LIN {X 0.106,Y -461.475,Z 275.770,A 0.000,B 0.000,C 90.000,E1 174.546} C_DIS
LIN {X -0.187,Y -461.115,Z 275.757,A 0.000,B 0.000,C 90.000,E1 172.356} C_DIS
LIN {X -0.159,Y -461.008,Z 275.747,A 0.000,B 0.000,C 90.000,E1 170.443} C_DIS
LIN {X 0.102,Y -461.301,Z 275.729,A 0.000,B 0.000,C 90.000,E1 167.229} C_DIS
LIN {X -0.019,Y -461.894,Z 275.715,A 0.000,B 0.000,C 90.000,E1 164.700} C_DIS
LIN {X 0.096,Y -462.800,Z 275.704,A 0.000,B 0.000,C 90.000,E1 162.779} C_DIS
LIN {X 0.096,Y -464.462,Z 275.690,A 0.000,B 0.000,C 90.000,E1 160.242} C_DIS
LIN {X 0.032,Y -466.538,Z 275.676,A 0.000,B 0.000,C 90.000,E1 157.720} C_DIS
LIN {X -0.223,Y -469.021,Z 275.662,A 0.000,B 0.000,C 90.000,E1 155.229} C_DIS
LIN {X -0.022,Y -472.104,Z 275.648,A 0.000,B 0.000,C 90.000,E1 152.692} C_DIS
LIN {X -0.131,Y -475.650,Z 275.634,A 0.000,B 0.000,C 90.000,E1 150.205} C_DIS
LIN {X -0.045,Y -478.598,Z 275.624,A 0.000,B 0.000,C 90.000,E1 148.329} C_DIS
LIN {X -0.298,Y -481.651,Z 275.614,A 0.000,B 0.000,C 90.000,E1 146.501} C_DIS
LIN {X 0.056,Y -484.820,Z 275.603,A 0.000,B 0.000,C 90.000,E1 144.609} C_DIS
LIN {X 0.261,Y -487.499,Z 275.595,A 0.000,B 0.000,C 90.000,E1 143.050} C_DIS
LIN {X 0.286,Y -489.476,Z 275.588,A 0.000,B 0.000,C 90.000,E1 141.823} C_DIS
LIN {X -0.203,Y -491.853,Z 275.580,A 0.000,B 0.000,C 90.000,E1 140.356} C_DIS
LIN {X 0.343,Y -493.148,Z 275.575,A 0.000,B 0.000,C 90.000,E1 139.380} C_DIS
LIN {X -0.317,Y -494.714,Z 275.568,A 0.000,B 0.000,C 90.000,E1 138.243} C_DIS
LIN {X -0.109,Y -495.734,Z 275.563,A 0.000,B 0.000,C 90.000,E1 137.310} C_DIS
LIN {X 0.299,Y -496.570,Z 275.556,A 0.000,B 0.000,C 90.000,E1 136.053} C_DIS
LIN {X 0.170,Y -497.012,Z 275.551,A 0.000,B 0.000,C 90.000,E1 135.162} C_DIS
LIN {X 0.047,Y -497.231,Z 275.546,A 0.000,B 0.000,C 90.000,E1 134.271} C_DIS
LIN {X -0.078,Y -497.156,Z 275.541,A 0.000,B 0.000,C 90.000,E1 133.380} C_DIS
LIN {X 0.158,Y -496.887,Z 275.536,A 0.000,B 0.000,C 90.000,E1 132.447} C_DIS
LIN {X 0.060,Y -496.384,Z 275.531,A 0.000,B 0.000,C 90.000,E1 131.553} C_DIS
LIN {X 0.286,Y -495.608,Z 275.526,A 0.000,B 0.000,C 90.000,E1 130.620} C_DIS
LIN {X 0.206,Y -493.919,Z 275.517,A 0.000,B 0.000,C 90.000,E1 129.116} C_DIS
LIN {X -0.074,Y -492.320,Z 275.511,A 0.000,B 0.000,C 90.000,E1 127.935} C_DIS
LIN {X 0.010,Y -490.558,Z 275.504,A 0.000,B 0.000,C 90.000,E1 126.710} C_DIS
LIN {X -0.223,Y -488.595,Z 275.497,A 0.000,B 0.000,C 90.000,E1 125.518} C_DIS
LIN {X -0.079,Y -486.458,Z 275.490,A 0.000,B 0.000,C 90.000,E1 124.278} C_DIS
LIN {X 0.035,Y -484.194,Z 275.484,A 0.000,B 0.000,C 90.000,E1 123.038} C_DIS
LIN {X -0.120,Y -480.685,Z 275.473,A 0.000,B 0.000,C 90.000,E1 121.209} C_DIS
LIN {X -0.152,Y -477.882,Z 275.465,A 0.000,B 0.000,C 90.000,E1 119.667} C_DIS
LIN {X 0.122,Y -474.366,Z 275.454,A 0.000,B 0.000,C 90.000,E1 117.769} C_DIS
LIN {X -0.118,Y -470.895,Z 275.444,A 0.000,B 0.000,C 90.000,E1 115.924} C_DIS
LIN {X 0.129,Y -466.736,Z 275.432,A 0.000,B 0.000,C 90.000,E1 113.695} C_DIS
LIN {X 0.132,Y -462.745,Z 275.419,A 0.000,B 0.000,C 90.000,E1 111.482} C_DIS
LIN {X -0.070,Y -458.602,Z 275.406,A 0.000,B 0.000,C 90.000,E1 109.087} C_DIS
LIN {X -0.110,Y -458.603,Z 275.406,A 0.000,B 0.000,C 90.000,E1 109.087} C_DIS
LIN {X -0.033,Y -467.907,Z 275.382,A 0.000,B 0.000,C 90.000,E1 104.828} C_DIS
LIN {X -0.006,Y -475.477,Z 275.358,A 0.000,B 0.000,C 90.000,E1 100.433} C_DIS
LIN {X -0.168,Y -476.121,Z 275.356,A 0.000,B 0.000,C 90.000,E1 100.141} C_DIS
LIN {X 0.115,Y -482.038,Z 275.330,A 0.000,B 0.000,C 90.000,E1 95.454} C_DIS
LIN {X -0.094,Y -485.472,Z 275.305,A 0.000,B 0.000,C 90.000,E1 90.859} C_DIS
LIN {X 0.147,Y -485.627,Z 275.293,A 0.000,B 0.000,C 90.000,E1 88.682} C_DIS
LIN {X -0.061,Y -486.385,Z 275.281,A 0.000,B 0.000,C 90.000,E1 86.560} C_DIS
LIN {X -0.236,Y -486.364,Z 275.279,A 0.000,B 0.000,C 90.000,E1 86.274} C_DIS
LIN {X -0.149,Y -484.689,Z 275.254,A 0.000,B 0.000,C 90.000,E1 81.659} C_DIS
LIN {X -0.134,Y -483.698,Z 275.249,A 0.000,B 0.000,C 90.000,E1 80.735} C_DIS
LIN {X 0.231,Y -480.628,Z 275.228,A 0.000,B 0.000,C 90.000,E1 76.992} C_DIS
LIN {X 0.088,Y -480.308,Z 275.226,A 0.000,B 0.000,C 90.000,E1 76.700} C_DIS
LIN {X -0.008,Y -474.127,Z 275.200,A 0.000,B 0.000,C 90.000,E1 72.054} C_DIS
LIN {X 0.081,Y -470.775,Z 275.191,A 0.000,B 0.000,C 90.000,E1 70.315} C_DIS
LIN {X 0.041,Y -470.787,Z 275.191,A 0.000,B 0.000,C 90.000,E1 70.315} C_DIS
LIN {X 0.174,Y -475.073,Z 275.181,A 0.000,B 0.000,C 90.000,E1 68.592} C_DIS
LIN {X 0.045,Y -479.937,Z 275.171,A 0.000,B 0.000,C 90.000,E1 66.741} C_DIS
LIN {X -0.231,Y -484.082,Z 275.162,A 0.000,B 0.000,C 90.000,E1 65.229} C_DIS
LIN {X -0.207,Y -489.044,Z 275.152,A 0.000,B 0.000,C 90.000,E1 63.384} C_DIS
LIN {X -0.125,Y -492.508,Z 275.145,A 0.000,B 0.000,C 90.000,E1 62.153} C_DIS
LIN {X -0.121,Y -497.684,Z 275.135,A 0.000,B 0.000,C 90.000,E1 60.333} C_DIS
LIN {X 0.200,Y -502.127,Z 275.127,A 0.000,B 0.000,C 90.000,E1 58.791} C_DIS
LIN {X -0.088,Y -506.507,Z 275.118,A 0.000,B 0.000,C 90.000,E1 57.327} C_DIS
LIN {X 0.160,Y -511.641,Z 275.109,A 0.000,B 0.000,C 90.000,E1 55.515} C_DIS
LIN {X 0.034,Y -514.022,Z 275.104,A 0.000,B 0.000,C 90.000,E1 54.642} C_DIS
LIN {X -0.019,Y -517.786,Z 275.095,A 0.000,B 0.000,C 90.000,E1 53.176} C_DIS
LIN {X 0.158,Y -520.628,Z 275.089,A 0.000,B 0.000,C 90.000,E1 51.984} C_DIS
LIN {X 0.235,Y -523.806,Z 275.081,A 0.000,B 0.000,C 90.000,E1 50.517} C_DIS
LIN {X 0.002,Y -526.034,Z 275.074,A 0.000,B 0.000,C 90.000,E1 49.380} C_DIS
LIN {X -0.197,Y -528.029,Z 275.068,A 0.000,B 0.000,C 90.000,E1 48.243} C_DIS
LIN {X -0.016,Y -529.645,Z 275.062,A 0.000,B 0.000,C 90.000,E1 47.067} C_DIS
LIN {X -0.143,Y -530.659,Z 275.057,A 0.000,B 0.000,C 90.000,E1 46.215} C_DIS
LIN {X 0.071,Y -531.764,Z 275.050,A 0.000,B 0.000,C 90.000,E1 45.040} C_DIS
LIN {X 0.300,Y -532.514,Z 275.044,A 0.000,B 0.000,C 90.000,E1 43.866} C_DIS
LIN {X -0.206,Y -532.946,Z 275.038,A 0.000,B 0.000,C 90.000,E1 42.771} C_DIS
LIN {X 0.045,Y -533.219,Z 275.031,A 0.000,B 0.000,C 90.000,E1 41.595} C_DIS
LIN {X -0.046,Y -533.229,Z 275.026,A 0.000,B 0.000,C 90.000,E1 40.744} C_DIS
LIN {X 0.257,Y -532.998,Z 275.020,A 0.000,B 0.000,C 90.000,E1 39.564} C_DIS
LIN {X -0.182,Y -532.650,Z 275.015,A 0.000,B 0.000,C 90.000,E1 38.749} C_DIS
LIN {X -0.213,Y -531.943,Z 275.009,A 0.000,B 0.000,C 90.000,E1 37.604} C_DIS
LIN {X 0.066,Y -531.117,Z 275.002,A 0.000,B 0.000,C 90.000,E1 36.423} C_DIS
LIN {X -0.300,Y -530.099,Z 274.996,A 0.000,B 0.000,C 90.000,E1 35.311} C_DIS
LIN {X 0.036,Y -528.628,Z 274.988,A 0.000,B 0.000,C 90.000,E1 33.833} C_DIS
LIN {X -0.242,Y -527.016,Z 274.980,A 0.000,B 0.000,C 90.000,E1 32.418} C_DIS
LIN {X -0.136,Y -524.963,Z 274.970,A 0.000,B 0.000,C 90.000,E1 30.669} C_DIS
LIN {X -0.026,Y -523.238,Z 274.962,A 0.000,B 0.000,C 90.000,E1 29.205} C_DIS
LIN {X -0.150,Y -520.850,Z 274.951,A 0.000,B 0.000,C 90.000,E1 27.180} C_DIS
LIN {X 0.017,Y -518.220,Z 274.938,A 0.000,B 0.000,C 90.000,E1 24.823} C_DIS
LIN {X -0.110,Y -516.487,Z 274.928,A 0.000,B 0.000,C 90.000,E1 23.078} C_DIS
LIN {X -0.151,Y -514.491,Z 274.917,A 0.000,B 0.000,C 90.000,E1 21.025} C_DIS
LIN {X -0.135,Y -512.731,Z 274.905,A 0.000,B 0.000,C 90.000,E1 18.960} C_DIS
LIN {X 0.124,Y -510.971,Z 274.892,A 0.000,B 0.000,C 90.000,E1 16.567} C_DIS
LIN {X 0.283,Y -509.262,Z 274.877,A 0.000,B 0.000,C 90.000,E1 13.883} C_DIS
LIN {X 0.008,Y -507.973,Z 274.863,A 0.000,B 0.000,C 90.000,E1 11.243} C_DIS
LIN {X 0.096,Y -507.342,Z 274.851,A 0.000,B 0.000,C 90.000,E1 9.151} C_DIS
LIN {X -0.013,Y -506.961,Z 274.836,A 0.000,B 0.000,C 90.000,E1 6.486} C_DIS
LIN {X 0.194,Y -507.156,Z 274.821,A 0.000,B 0.000,C 90.000,E1 3.784} C_DIS
LIN {X -0.253,Y -507.978,Z 274.805,A 0.000,B 0.000,C 90.000,E1 0.859} C_DIS
LIN {X 0.066,Y -509.824,Z 274.787,A 0.000,B 0.000,C 90.000,E1 357.707} C_DIS
LIN {X -0.233,Y -512.446,Z 274.771,A 0.000,B 0.000,C 90.000,E1 354.780} C_DIS
LIN {X 0.058,Y -517.639,Z 274.748,A 0.000,B 0.000,C 90.000,E1 350.622} C_DIS
LIN {X 0.022,Y -522.854,Z 274.733,A 0.000,B 0.000,C 90.000,E1 347.993} C_DIS
LIN {X -0.230,Y -529.405,Z 274.719,A 0.000,B 0.000,C 90.000,E1 345.408} C_DIS
LIN {X -0.094,Y -534.660,Z 274.708,A 0.000,B 0.000,C 90.000,E1 343.378} C_DIS
LIN {X -0.116,Y -543.637,Z 274.690,A 0.000,B 0.000,C 90.000,E1 340.242} C_DIS
LIN {X -0.026,Y -550.953,Z 274.678,A 0.000,B 0.000,C 90.000,E1 337.975} C_DIS
LIN {X -0.107,Y -556.715,Z 274.668,A 0.000,B 0.000,C 90.000,E1 336.305} C_DIS
LIN {X 0.317,Y -565.535,Z 274.654,A 0.000,B 0.000,C 90.000,E1 333.768} C_DIS
LIN {X 0.002,Y -571.669,Z 274.645,A 0.000,B 0.000,C 90.000,E1 332.153} C_DIS
LIN {X 0.282,Y -574.685,Z 274.641,A 0.000,B 0.000,C 90.000,E1 331.307} C_DIS
LIN {X -0.212,Y -579.472,Z 274.633,A 0.000,B 0.000,C 90.000,E1 329.999} C_DIS
LIN {X 0.160,Y -584.103,Z 274.626,A 0.000,B 0.000,C 90.000,E1 328.614} C_DIS
LIN {X 0.074,Y -592.492,Z 274.612,A 0.000,B 0.000,C 90.000,E1 326.215} C_DIS
LIN {X 0.114,Y -599.456,Z 274.602,A 0.000,B 0.000,C 90.000,E1 324.356} C_DIS
LIN {X 0.018,Y -604.315,Z 274.595,A 0.000,B 0.000,C 90.000,E1 323.050} C_DIS
LIN {X 0.015,Y -608.859,Z 274.588,A 0.000,B 0.000,C 90.000,E1 321.743} C_DIS
LIN {X -0.100,Y -614.070,Z 274.579,A 0.000,B 0.000,C 90.000,E1 320.194} C_DIS
LIN {X 0.313,Y -616.511,Z 274.575,A 0.000,B 0.000,C 90.000,E1 319.380} C_DIS
LIN {X -0.133,Y -621.354,Z 274.566,A 0.000,B 0.000,C 90.000,E1 317.877} C_DIS
LIN {X 0.029,Y -625.262,Z 274.559,A 0.000,B 0.000,C 90.000,E1 316.581} C_DIS
LIN {X -0.289,Y -629.579,Z 274.550,A 0.000,B 0.000,C 90.000,E1 315.081} C_DIS
LIN {X 0.025,Y -633.123,Z 274.543,A 0.000,B 0.000,C 90.000,E1 313.785} C_DIS
LIN {X -0.043,Y -636.506,Z 274.536,A 0.000,B 0.000,C 90.000,E1 312.528} C_DIS
LIN {X 0.034,Y -638.981,Z 274.531,A 0.000,B 0.000,C 90.000,E1 311.515} C_DIS
LIN {X -0.188,Y -640.685,Z 274.527,A 0.000,B 0.000,C 90.000,E1 310.782} C_DIS
LIN {X -0.065,Y -642.601,Z 274.521,A 0.000,B 0.000,C 90.000,E1 309.769} C_DIS
LIN {X 0.163,Y -644.329,Z 274.515,A 0.000,B 0.000,C 90.000,E1 308.749} C_DIS
LIN {X 0.418,Y -645.937,Z 274.510,A 0.000,B 0.000,C 90.000,E1 307.729} C_DIS
LIN {X -0.213,Y -647.265,Z 274.504,A 0.000,B 0.000,C 90.000,E1 306.790} C_DIS
LIN {X -0.263,Y -647.848,Z 274.502,A 0.000,B 0.000,C 90.000,E1 306.297} C_DIS
LIN {X 0.123,Y -648.442,Z 274.497,A 0.000,B 0.000,C 90.000,E1 305.518} C_DIS
LIN {X 0.042,Y -648.789,Z 274.492,A 0.000,B 0.000,C 90.000,E1 304.532} C_DIS
LIN {X -0.400,Y -648.941,Z 274.486,A 0.000,B 0.000,C 90.000,E1 303.579} C_DIS
LIN {X -0.015,Y -648.810,Z 274.482,A 0.000,B 0.000,C 90.000,E1 302.801} C_DIS
LIN {X 0.139,Y -648.623,Z 274.480,A 0.000,B 0.000,C 90.000,E1 302.291} C_DIS
LIN {X 0.170,Y -647.994,Z 274.475,A 0.000,B 0.000,C 90.000,E1 301.544} C_DIS
LIN {X 0.192,Y -646.986,Z 274.471,A 0.000,B 0.000,C 90.000,E1 300.797} C_DIS
LIN {X 0.274,Y -645.292,Z 274.466,A 0.000,B 0.000,C 90.000,E1 299.795} C_DIS
LIN {X -0.059,Y -643.650,Z 274.462,A 0.000,B 0.000,C 90.000,E1 299.077} C_DIS
LIN {X -0.267,Y -640.659,Z 274.455,A 0.000,B 0.000,C 90.000,E1 297.847} C_DIS
LIN {X 0.048,Y -637.516,Z 274.448,A 0.000,B 0.000,C 90.000,E1 296.565} C_DIS
LIN {X -0.265,Y -634.203,Z 274.441,A 0.000,B 0.000,C 90.000,E1 295.335} C_DIS
LIN {X 0.270,Y -630.167,Z 274.432,A 0.000,B 0.000,C 90.000,E1 293.770} C_DIS
LIN {X -0.090,Y -625.441,Z 274.422,A 0.000,B 0.000,C 90.000,E1 292.025} C_DIS
LIN {X 0.023,Y -621.631,Z 274.414,A 0.000,B 0.000,C 90.000,E1 290.482} C_DIS
LIN {X 0.145,Y -616.643,Z 274.402,A 0.000,B 0.000,C 90.000,E1 288.417} C_DIS
LIN {X -0.221,Y -610.483,Z 274.387,A 0.000,B 0.000,C 90.000,E1 285.607} C_DIS
LIN {X -0.329,Y -606.566,Z 274.375,A 0.000,B 0.000,C 90.000,E1 283.536} C_DIS
LIN {X 0.192,Y -601.572,Z 274.356,A 0.000,B 0.000,C 90.000,E1 280.084} C_DIS
LIN {X 0.285,Y -598.493,Z 274.340,A 0.000,B 0.000,C 90.000,E1 277.182} C_DIS
LIN {X 0.294,Y -597.095,Z 274.330,A 0.000,B 0.000,C 90.000,E1 275.334} C_DIS
LIN {X -0.096,Y -595.883,Z 274.314,A 0.000,B 0.000,C 90.000,E1 272.465} C_DIS
LIN {X 0.177,Y -595.641,Z 274.300,A 0.000,B 0.000,C 90.000,E1 270.057} C_DIS
LIN {X -0.061,Y -596.591,Z 274.283,A 0.000,B 0.000,C 90.000,E1 266.906} C_DIS
LIN {X 0.203,Y -598.718,Z 274.267,A 0.000,B 0.000,C 90.000,E1 263.976} C_DIS
LIN {X 0.242,Y -601.248,Z 274.254,A 0.000,B 0.000,C 90.000,E1 261.602} C_DIS
LIN {X -0.117,Y -604.430,Z 274.240,A 0.000,B 0.000,C 90.000,E1 259.275} C_DIS
LIN {X -0.004,Y -607.729,Z 274.229,A 0.000,B 0.000,C 90.000,E1 257.173} C_DIS
LIN {X -0.112,Y -609.781,Z 274.222,A 0.000,B 0.000,C 90.000,E1 255.880} C_DIS
LIN {X 0.213,Y -611.384,Z 274.216,A 0.000,B 0.000,C 90.000,E1 254.810} C_DIS
LIN {X -0.026,Y -612.875,Z 274.210,A 0.000,B 0.000,C 90.000,E1 253.795} C_DIS
LIN {X 0.001,Y -613.682,Z 274.206,A 0.000,B 0.000,C 90.000,E1 253.015} C_DIS
LIN {X -0.209,Y -614.439,Z 274.200,A 0.000,B 0.000,C 90.000,E1 252.000} C_DIS
LIN {X -0.220,Y -614.992,Z 274.194,A 0.000,B 0.000,C 90.000,E1 250.967} C_DIS
LIN {X -0.220,Y -615.197,Z 274.188,A 0.000,B 0.000,C 90.000,E1 249.934} C_DIS
LIN {X 0.032,Y -615.152,Z 274.184,A 0.000,B 0.000,C 90.000,E1 249.135} C_DIS
LIN {X 0.057,Y -614.841,Z 274.180,A 0.000,B 0.000,C 90.000,E1 248.358} C_DIS
LIN {X -0.305,Y -613.992,Z 274.174,A 0.000,B 0.000,C 90.000,E1 247.358} C_DIS
LIN {X 0.168,Y -613.160,Z 274.170,A 0.000,B 0.000,C 90.000,E1 246.538} C_DIS
LIN {X -0.173,Y -612.026,Z 274.165,A 0.000,B 0.000,C 90.000,E1 245.793} C_DIS
LIN {X 0.281,Y -610.653,Z 274.161,A 0.000,B 0.000,C 90.000,E1 244.973} C_DIS
LIN {X 0.169,Y -609.068,Z 274.157,A 0.000,B 0.000,C 90.000,E1 244.204} C_DIS
LIN {X 0.000,Y -606.607,Z 274.151,A 0.000,B 0.000,C 90.000,E1 243.179} C_DIS
LIN {X -0.261,Y -603.335,Z 274.144,A 0.000,B 0.000,C 90.000,E1 241.897} C_DIS
LIN {X -0.225,Y -600.583,Z 274.138,A 0.000,B 0.000,C 90.000,E1 240.845} C_DIS
LIN {X -0.309,Y -597.013,Z 274.131,A 0.000,B 0.000,C 90.000,E1 239.537} C_DIS
LIN {X -0.059,Y -593.951,Z 274.125,A 0.000,B 0.000,C 90.000,E1 238.456} C_DIS
LIN {X 0.034,Y -589.964,Z 274.117,A 0.000,B 0.000,C 90.000,E1 237.120} C_DIS
LIN {X 0.070,Y -584.802,Z 274.108,A 0.000,B 0.000,C 90.000,E1 235.515} C_DIS
LIN {X 0.174,Y -578.793,Z 274.098,A 0.000,B 0.000,C 90.000,E1 233.623} C_DIS
LIN {X 0.165,Y -574.664,Z 274.091,A 0.000,B 0.000,C 90.000,E1 232.271} C_DIS
LIN {X 0.248,Y -568.723,Z 274.080,A 0.000,B 0.000,C 90.000,E1 230.356} C_DIS
LIN {X -0.141,Y -565.383,Z 274.074,A 0.000,B 0.000,C 90.000,E1 229.299} C_DIS
LIN {X -0.017,Y -560.214,Z 274.065,A 0.000,B 0.000,C 90.000,E1 227.634} C_DIS
LIN {X -0.043,Y -555.005,Z 274.055,A 0.000,B 0.000,C 90.000,E1 225.972} C_DIS
LIN {X 0.208,Y -549.775,Z 274.046,A 0.000,B 0.000,C 90.000,E1 224.271} C_DIS
LIN {X -0.067,Y -546.213,Z 274.040,A 0.000,B 0.000,C 90.000,E1 223.176} C_DIS
LIN {X 0.018,Y -540.950,Z 274.030,A 0.000,B 0.000,C 90.000,E1 221.472} C_DIS
LIN {X 0.026,Y -537.498,Z 274.024,A 0.000,B 0.000,C 90.000,E1 220.334} C_DIS
LIN {X -0.030,Y -531.353,Z 274.013,A 0.000,B 0.000,C 90.000,E1 218.338} C_DIS
LIN {X 0.220,Y -527.040,Z 274.005,A 0.000,B 0.000,C 90.000,E1 216.870} C_DIS
LIN {X 0.023,Y -521.959,Z 273.995,A 0.000,B 0.000,C 90.000,E1 215.152} C_DIS
LIN {X 0.204,Y -516.165,Z 273.984,A 0.000,B 0.000,C 90.000,E1 213.086} C_DIS
LIN {X 0.051,Y -511.394,Z 273.974,A 0.000,B 0.000,C 90.000,E1 211.337} C_DIS
LIN {X -0.132,Y -506.033,Z 273.963,A 0.000,B 0.000,C 90.000,E1 209.283} C_DIS
LIN {X -0.021,Y -500.950,Z 273.951,A 0.000,B 0.000,C 90.000,E1 207.180} C_DIS
LIN {X -0.010,Y -495.618,Z 273.938,A 0.000,B 0.000,C 90.000,E1 204.771} C_DIS
LIN {X 0.096,Y -490.640,Z 273.924,A 0.000,B 0.000,C 90.000,E1 202.333} C_DIS
LIN {X 0.162,Y -485.479,Z 273.909,A 0.000,B 0.000,C 90.000,E1 199.577} C_DIS
LIN {X -0.106,Y -481.804,Z 273.897,A 0.000,B 0.000,C 90.000,E1 197.457} C_DIS
LIN {X 0.035,Y -479.893,Z 273.890,A 0.000,B 0.000,C 90.000,E1 196.205} C_DIS
LIN {X 0.063,Y -475.812,Z 273.875,A 0.000,B 0.000,C 90.000,E1 193.411} C_DIS
LIN {X 0.121,Y -473.487,Z 273.864,A 0.000,B 0.000,C 90.000,E1 191.535} C_DIS
LIN {X -0.108,Y -470.110,Z 273.849,A 0.000,B 0.000,C 90.000,E1 188.746} C_DIS
LIN {X -0.075,Y -467.869,Z 273.836,A 0.000,B 0.000,C 90.000,E1 186.543} C_DIS
LIN {X 0.199,Y -465.790,Z 273.824,A 0.000,B 0.000,C 90.000,E1 184.302} C_DIS
LIN {X -0.064,Y -464.101,Z 273.812,A 0.000,B 0.000,C 90.000,E1 182.121} C_DIS
LIN {X -0.177,Y -462.406,Z 273.798,A 0.000,B 0.000,C 90.000,E1 179.599} C_DIS
LIN {X 0.169,Y -461.460,Z 273.787,A 0.000,B 0.000,C 90.000,E1 177.650} C_DIS
LIN {X 0.219,Y -460.436,Z 273.771,A 0.000,B 0.000,C 90.000,E1 174.780} C_DIS
LIN {X 0.127,Y -460.036,Z 273.757,A 0.000,B 0.000,C 90.000,E1 172.243} C_DIS
LIN {X 0.125,Y -459.934,Z 273.746,A 0.000,B 0.000,C 90.000,E1 170.330} C_DIS
LIN {X -0.113,Y -460.277,Z 273.729,A 0.000,B 0.000,C 90.000,E1 167.173} C_DIS
LIN {X 0.163,Y -460.716,Z 273.718,A 0.000,B 0.000,C 90.000,E1 165.227} C_DIS
LIN {X 0.174,Y -461.984,Z 273.702,A 0.000,B 0.000,C 90.000,E1 162.362} C_DIS
LIN {X 0.143,Y -463.762,Z 273.688,A 0.000,B 0.000,C 90.000,E1 159.826} C_DIS
LIN {X 0.045,Y -465.915,Z 273.674,A 0.000,B 0.000,C 90.000,E1 157.305} C_DIS
LIN {X 0.006,Y -468.138,Z 273.662,A 0.000,B 0.000,C 90.000,E1 155.101} C_DIS
LIN {X -0.237,Y -471.251,Z 273.648,A 0.000,B 0.000,C 90.000,E1 152.615} C_DIS
LIN {X 0.046,Y -474.825,Z 273.634,A 0.000,B 0.000,C 90.000,E1 150.078} C_DIS
LIN {X -0.097,Y -478.255,Z 273.622,A 0.000,B 0.000,C 90.000,E1 147.916} C_DIS
LIN {X 0.105,Y -480.805,Z 273.613,A 0.000,B 0.000,C 90.000,E1 146.342} C_DIS
LIN {X -0.043,Y -483.480,Z 273.605,A 0.000,B 0.000,C 90.000,E1 144.815} C_DIS
LIN {X 0.138,Y -486.143,Z 273.596,A 0.000,B 0.000,C 90.000,E1 143.256} C_DIS
LIN {X -0.022,Y -488.622,Z 273.587,A 0.000,B 0.000,C 90.000,E1 141.743} C_DIS
LIN {X 0.014,Y -490.537,Z 273.581,A 0.000,B 0.000,C 90.000,E1 140.517} C_DIS
LIN {X 0.010,Y -492.235,Z 273.574,A 0.000,B 0.000,C 90.000,E1 139.299} C_DIS
LIN {X 0.034,Y -493.774,Z 273.567,A 0.000,B 0.000,C 90.000,E1 138.081} C_DIS
LIN {X 0.233,Y -494.749,Z 273.562,A 0.000,B 0.000,C 90.000,E1 137.148} C_DIS
LIN {X -0.074,Y -495.588,Z 273.555,A 0.000,B 0.000,C 90.000,E1 135.972} C_DIS
LIN {X -0.214,Y -495.972,Z 273.550,A 0.000,B 0.000,C 90.000,E1 135.081} C_DIS
LIN {X -0.003,Y -496.151,Z 273.545,A 0.000,B 0.000,C 90.000,E1 134.150} C_DIS
LIN {X -0.123,Y -496.078,Z 273.540,A 0.000,B 0.000,C 90.000,E1 133.257} C_DIS
LIN {X 0.104,Y -495.802,Z 273.535,A 0.000,B 0.000,C 90.000,E1 132.324} C_DIS
LIN {X -0.044,Y -495.264,Z 273.530,A 0.000,B 0.000,C 90.000,E1 131.434} C_DIS
LIN {X -0.159,Y -494.478,Z 273.525,A 0.000,B 0.000,C 90.000,E1 130.539} C_DIS
LIN {X 0.123,Y -492.800,Z 273.517,A 0.000,B 0.000,C 90.000,E1 128.991} C_DIS
LIN {X -0.168,Y -491.210,Z 273.510,A 0.000,B 0.000,C 90.000,E1 127.810} C_DIS
LIN {X -0.097,Y -489.447,Z 273.503,A 0.000,B 0.000,C 90.000,E1 126.583} C_DIS
LIN {X 0.106,Y -487.980,Z 273.498,A 0.000,B 0.000,C 90.000,E1 125.644} C_DIS
LIN {X 0.235,Y -485.865,Z 273.491,A 0.000,B 0.000,C 90.000,E1 124.405} C_DIS
LIN {X 0.153,Y -483.051,Z 273.483,A 0.000,B 0.000,C 90.000,E1 122.880} C_DIS
LIN {X -0.039,Y -479.596,Z 273.473,A 0.000,B 0.000,C 90.000,E1 121.052} C_DIS
LIN {X 0.079,Y -476.756,Z 273.464,A 0.000,B 0.000,C 90.000,E1 119.489} C_DIS
LIN {X -0.265,Y -473.866,Z 273.455,A 0.000,B 0.000,C 90.000,E1 117.975} C_DIS
LIN {X 0.122,Y -470.384,Z 273.445,A 0.000,B 0.000,C 90.000,E1 116.052} C_DIS
LIN {X -0.204,Y -466.818,Z 273.434,A 0.000,B 0.000,C 90.000,E1 114.207} C_DIS
LIN {X 0.114,Y -463.898,Z 273.426,A 0.000,B 0.000,C 90.000,E1 112.589} C_DIS
LIN {X -0.155,Y -461.661,Z 273.419,A 0.000,B 0.000,C 90.000,E1 111.354} C_DIS
LIN {X 0.218,Y -458.203,Z 273.407,A 0.000,B 0.000,C 90.000,E1 109.268} C_DIS
LIN {X 0.178,Y -458.203,Z 273.407,A 0.000,B 0.000,C 90.000,E1 109.268} C_DIS
LIN {X -0.084,Y -466.797,Z 273.385,A 0.000,B 0.000,C 90.000,E1 105.300} C_DIS
LIN {X 0.168,Y -467.589,Z 273.383,A 0.000,B 0.000,C 90.000,E1 104.954} C_DIS
LIN {X -0.100,Y -468.589,Z 273.380,A 0.000,B 0.000,C 90.000,E1 104.356} C_DIS
LIN {X 0.127,Y -475.819,Z 273.357,A 0.000,B 0.000,C 90.000,E1 100.254} C_DIS
LIN {X -0.035,Y -476.313,Z 273.355,A 0.000,B 0.000,C 90.000,E1 99.962} C_DIS
LIN {X -0.088,Y -481.802,Z 273.331,A 0.000,B 0.000,C 90.000,E1 95.625} C_DIS
LIN {X 0.239,Y -482.174,Z 273.330,A 0.000,B 0.000,C 90.000,E1 95.277} C_DIS
LIN {X 0.173,Y -485.316,Z 273.306,A 0.000,B 0.000,C 90.000,E1 90.974} C_DIS
LIN {X -0.002,Y -485.536,Z 273.304,A 0.000,B 0.000,C 90.000,E1 90.688} C_DIS
LIN {X 0.205,Y -486.323,Z 273.282,A 0.000,B 0.000,C 90.000,E1 86.674} C_DIS
LIN {X -0.145,Y -486.299,Z 273.278,A 0.000,B 0.000,C 90.000,E1 86.102} C_DIS
LIN {X 0.059,Y -484.695,Z 273.254,A 0.000,B 0.000,C 90.000,E1 81.781} C_DIS
LIN {X -0.072,Y -484.590,Z 273.253,A 0.000,B 0.000,C 90.000,E1 81.489} C_DIS
LIN {X -0.192,Y -480.526,Z 273.227,A 0.000,B 0.000,C 90.000,E1 76.881} C_DIS
LIN {X 0.171,Y -474.277,Z 273.201,A 0.000,B 0.000,C 90.000,E1 72.181} C_DIS
LIN {X 0.139,Y -473.831,Z 273.199,A 0.000,B 0.000,C 90.000,E1 71.873} C_DIS
LIN {X 0.017,Y -470.434,Z 273.190,A 0.000,B 0.000,C 90.000,E1 70.134} C_DIS
LIN {X 0.138,Y -470.434,Z 273.190,A 0.000,B 0.000,C 90.000,E1 70.115} C_DIS
LIN {X -0.138,Y -474.675,Z 273.180,A 0.000,B 0.000,C 90.000,E1 68.465} C_DIS
LIN {X -0.277,Y -479.528,Z 273.170,A 0.000,B 0.000,C 90.000,E1 66.613} C_DIS
LIN {X -0.123,Y -483.664,Z 273.161,A 0.000,B 0.000,C 90.000,E1 65.049} C_DIS
LIN {X 0.120,Y -489.506,Z 273.149,A 0.000,B 0.000,C 90.000,E1 62.871} C_DIS
LIN {X 0.057,Y -494.698,Z 273.139,A 0.000,B 0.000,C 90.000,E1 61.051} C_DIS
LIN {X -0.075,Y -499.947,Z 273.129,A 0.000,B 0.000,C 90.000,E1 59.253} C_DIS
LIN {X 0.028,Y -504.372,Z 273.121,A 0.000,B 0.000,C 90.000,E1 57.740} C_DIS
LIN {X 0.108,Y -506.951,Z 273.116,A 0.000,B 0.000,C 90.000,E1 56.834} C_DIS
LIN {X -0.250,Y -511.184,Z 273.108,A 0.000,B 0.000,C 90.000,E1 55.388} C_DIS
LIN {X -0.167,Y -514.288,Z 273.101,A 0.000,B 0.000,C 90.000,E1 54.196} C_DIS
LIN {X -0.042,Y -517.281,Z 273.094,A 0.000,B 0.000,C 90.000,E1 53.004} C_DIS
LIN {X 0.028,Y -520.053,Z 273.088,A 0.000,B 0.000,C 90.000,E1 51.823} C_DIS
LIN {X 0.097,Y -523.167,Z 273.080,A 0.000,B 0.000,C 90.000,E1 50.356} C_DIS
LIN {X -0.142,Y -525.362,Z 273.073,A 0.000,B 0.000,C 90.000,E1 49.218} C_DIS
LIN {X 0.041,Y -527.271,Z 273.067,A 0.000,B 0.000,C 90.000,E1 48.038} C_DIS
LIN {X -0.180,Y -528.847,Z 273.061,A 0.000,B 0.000,C 90.000,E1 46.905} C_DIS
LIN {X 0.015,Y -530.073,Z 273.054,A 0.000,B 0.000,C 90.000,E1 45.729} C_DIS
LIN {X 0.261,Y -530.830,Z 273.049,A 0.000,B 0.000,C 90.000,E1 44.838} C_DIS
LIN {X 0.100,Y -531.492,Z 273.043,A 0.000,B 0.000,C 90.000,E1 43.704} C_DIS
LIN {X 0.330,Y -531.866,Z 273.037,A 0.000,B 0.000,C 90.000,E1 42.528} C_DIS
LIN {X 0.228,Y -532.055,Z 273.032,A 0.000,B 0.000,C 90.000,E1 41.676} C_DIS
LIN {X 0.126,Y -532.076,Z 273.027,A 0.000,B 0.000,C 90.000,E1 40.825} C_DIS
LIN {X 0.003,Y -531.842,Z 273.021,A 0.000,B 0.000,C 90.000,E1 39.688} C_DIS
LIN {X -0.037,Y -531.480,Z 273.016,A 0.000,B 0.000,C 90.000,E1 38.830} C_DIS
LIN {X 0.227,Y -530.603,Z 273.008,A 0.000,B 0.000,C 90.000,E1 37.363} C_DIS
LIN {X 0.181,Y -529.962,Z 273.003,A 0.000,B 0.000,C 90.000,E1 36.503} C_DIS
LIN {X -0.200,Y -528.928,Z 272.997,A 0.000,B 0.000,C 90.000,E1 35.391} C_DIS
LIN {X 0.118,Y -527.423,Z 272.989,A 0.000,B 0.000,C 90.000,E1 33.913} C_DIS
LIN {X 0.104,Y -525.770,Z 272.980,A 0.000,B 0.000,C 90.000,E1 32.467} C_DIS
LIN {X 0.173,Y -523.687,Z 272.971,A 0.000,B 0.000,C 90.000,E1 30.718} C_DIS
LIN {X -0.072,Y -521.574,Z 272.961,A 0.000,B 0.000,C 90.000,E1 28.999} C_DIS
LIN {X -0.152,Y -519.530,Z 272.951,A 0.000,B 0.000,C 90.000,E1 27.257} C_DIS
LIN {X -0.015,Y -516.875,Z 272.938,A 0.000,B 0.000,C 90.000,E1 24.899} C_DIS
LIN {X 0.038,Y -515.125,Z 272.929,A 0.000,B 0.000,C 90.000,E1 23.131} C_DIS
LIN {X -0.229,Y -513.110,Z 272.917,A 0.000,B 0.000,C 90.000,E1 21.099} C_DIS
LIN {X -0.237,Y -511.332,Z 272.906,A 0.000,B 0.000,C 90.000,E1 19.033} C_DIS
LIN {X 0.139,Y -509.528,Z 272.892,A 0.000,B 0.000,C 90.000,E1 16.622} C_DIS
LIN {X 0.120,Y -507.771,Z 272.878,A 0.000,B 0.000,C 90.000,E1 13.953} C_DIS
LIN {X -0.087,Y -506.455,Z 272.863,A 0.000,B 0.000,C 90.000,E1 11.299} C_DIS
LIN {X -0.096,Y -505.703,Z 272.850,A 0.000,B 0.000,C 90.000,E1 8.916} C_DIS
LIN {X -0.205,Y -505.390,Z 272.836,A 0.000,B 0.000,C 90.000,E1 6.543} C_DIS
LIN {X -0.054,Y -505.528,Z 272.821,A 0.000,B 0.000,C 90.000,E1 3.841} C_DIS
LIN {X -0.055,Y -506.327,Z 272.805,A 0.000,B 0.000,C 90.000,E1 0.859} C_DIS
LIN {X 0.023,Y -508.163,Z 272.787,A 0.000,B 0.000,C 90.000,E1 357.707} C_DIS
LIN {X 0.170,Y -510.756,Z 272.771,A 0.000,B 0.000,C 90.000,E1 354.723} C_DIS
LIN {X 0.042,Y -514.169,Z 272.754,A 0.000,B 0.000,C 90.000,E1 351.781} C_DIS
LIN {X -0.156,Y -516.484,Z 272.746,A 0.000,B 0.000,C 90.000,E1 350.330} C_DIS
LIN {X -0.230,Y -521.210,Z 272.733,A 0.000,B 0.000,C 90.000,E1 347.993} C_DIS
LIN {X 0.108,Y -527.817,Z 272.719,A 0.000,B 0.000,C 90.000,E1 345.338} C_DIS
LIN {X -0.142,Y -531.533,Z 272.711,A 0.000,B 0.000,C 90.000,E1 343.921} C_DIS
LIN {X 0.214,Y -537.062,Z 272.699,A 0.000,B 0.000,C 90.000,E1 341.873} C_DIS
LIN {X 0.225,Y -545.747,Z 272.684,A 0.000,B 0.000,C 90.000,E1 339.028} C_DIS
LIN {X -0.204,Y -552.344,Z 272.673,A 0.000,B 0.000,C 90.000,E1 337.102} C_DIS
LIN {X 0.186,Y -557.203,Z 272.665,A 0.000,B 0.000,C 90.000,E1 335.665} C_DIS
LIN {X -0.122,Y -566.171,Z 272.651,A 0.000,B 0.000,C 90.000,E1 333.204} C_DIS
LIN {X 0.006,Y -571.342,Z 272.643,A 0.000,B 0.000,C 90.000,E1 331.820} C_DIS
LIN {X -0.039,Y -576.213,Z 272.636,A 0.000,B 0.000,C 90.000,E1 330.461} C_DIS
LIN {X -0.220,Y -580.928,Z 272.628,A 0.000,B 0.000,C 90.000,E1 329.125} C_DIS
LIN {X -0.142,Y -586.445,Z 272.619,A 0.000,B 0.000,C 90.000,E1 327.502} C_DIS
LIN {X -0.143,Y -595.222,Z 272.606,A 0.000,B 0.000,C 90.000,E1 325.102} C_DIS
LIN {X -0.178,Y -600.212,Z 272.599,A 0.000,B 0.000,C 90.000,E1 323.783} C_DIS
LIN {X -0.036,Y -604.007,Z 272.593,A 0.000,B 0.000,C 90.000,E1 322.718} C_DIS
LIN {X -0.056,Y -608.481,Z 272.586,A 0.000,B 0.000,C 90.000,E1 321.412} C_DIS
LIN {X 0.202,Y -613.606,Z 272.577,A 0.000,B 0.000,C 90.000,E1 319.828} C_DIS
LIN {X -0.297,Y -618.498,Z 272.568,A 0.000,B 0.000,C 90.000,E1 318.324} C_DIS
LIN {X -0.309,Y -620.925,Z 272.564,A 0.000,B 0.000,C 90.000,E1 317.553} C_DIS
LIN {X -0.012,Y -624.121,Z 272.558,A 0.000,B 0.000,C 90.000,E1 316.500} C_DIS
LIN {X 0.093,Y -628.467,Z 272.550,A 0.000,B 0.000,C 90.000,E1 314.960} C_DIS
LIN {X 0.057,Y -631.328,Z 272.544,A 0.000,B 0.000,C 90.000,E1 313.947} C_DIS
LIN {X -0.039,Y -634.714,Z 272.537,A 0.000,B 0.000,C 90.000,E1 312.690} C_DIS
LIN {X 0.118,Y -636.596,Z 272.533,A 0.000,B 0.000,C 90.000,E1 311.919} C_DIS
LIN {X 0.293,Y -638.347,Z 272.529,A 0.000,B 0.000,C 90.000,E1 311.148} C_DIS
LIN {X 0.070,Y -639.938,Z 272.525,A 0.000,B 0.000,C 90.000,E1 310.415} C_DIS
LIN {X 0.182,Y -641.808,Z 272.519,A 0.000,B 0.000,C 90.000,E1 309.402} C_DIS
LIN {X -0.091,Y -643.833,Z 272.512,A 0.000,B 0.000,C 90.000,E1 308.177} C_DIS
LIN {X 0.159,Y -645.299,Z 272.507,A 0.000,B 0.000,C 90.000,E1 307.156} C_DIS
LIN {X -0.001,Y -646.204,Z 272.502,A 0.000,B 0.000,C 90.000,E1 306.423} C_DIS
LIN {X -0.012,Y -646.832,Z 272.498,A 0.000,B 0.000,C 90.000,E1 305.678} C_DIS
LIN {X -0.109,Y -647.234,Z 272.493,A 0.000,B 0.000,C 90.000,E1 304.692} C_DIS
LIN {X -0.140,Y -647.394,Z 272.486,A 0.000,B 0.000,C 90.000,E1 303.452} C_DIS
LIN {X 0.231,Y -647.233,Z 272.482,A 0.000,B 0.000,C 90.000,E1 302.673} C_DIS
LIN {X 0.245,Y -646.794,Z 272.478,A 0.000,B 0.000,C 90.000,E1 301.926} C_DIS
LIN {X -0.158,Y -646.321,Z 272.475,A 0.000,B 0.000,C 90.000,E1 301.465} C_DIS
LIN {X -0.156,Y -645.275,Z 272.471,A 0.000,B 0.000,C 90.000,E1 300.718} C_DIS
LIN {X 0.066,Y -643.987,Z 272.466,A 0.000,B 0.000,C 90.000,E1 299.951} C_DIS
LIN {X 0.041,Y -642.415,Z 272.462,A 0.000,B 0.000,C 90.000,E1 299.205} C_DIS
LIN {X -0.188,Y -639.452,Z 272.455,A 0.000,B 0.000,C 90.000,E1 297.975} C_DIS
LIN {X 0.105,Y -636.302,Z 272.448,A 0.000,B 0.000,C 90.000,E1 296.693} C_DIS
LIN {X -0.227,Y -632.993,Z 272.441,A 0.000,B 0.000,C 90.000,E1 295.463} C_DIS
LIN {X 0.306,Y -628.273,Z 272.432,A 0.000,B 0.000,C 90.000,E1 293.643} C_DIS
LIN {X -0.101,Y -624.219,Z 272.423,A 0.000,B 0.000,C 90.000,E1 292.153} C_DIS
LIN {X -0.011,Y -620.386,Z 272.415,A 0.000,B 0.000,C 90.000,E1 290.610} C_DIS
LIN {X 0.085,Y -615.406,Z 272.403,A 0.000,B 0.000,C 90.000,E1 288.544} C_DIS
LIN {X -0.065,Y -609.747,Z 272.389,A 0.000,B 0.000,C 90.000,E1 285.969} C_DIS
LIN {X 0.020,Y -604.811,Z 272.374,A 0.000,B 0.000,C 90.000,E1 283.355} C_DIS
LIN {X 0.119,Y -600.941,Z 272.360,A 0.000,B 0.000,C 90.000,E1 280.725} C_DIS
LIN {X 0.275,Y -597.621,Z 272.344,A 0.000,B 0.000,C 90.000,E1 277.814} C_DIS
LIN {X -0.121,Y -595.911,Z 272.332,A 0.000,B 0.000,C 90.000,E1 275.739} C_DIS
LIN {X -0.294,Y -594.474,Z 272.314,A 0.000,B 0.000,C 90.000,E1 272.579} C_DIS
LIN {X -0.217,Y -594.245,Z 272.298,A 0.000,B 0.000,C 90.000,E1 269.656} C_DIS
LIN {X 0.233,Y -595.149,Z 272.283,A 0.000,B 0.000,C 90.000,E1 266.963} C_DIS
LIN {X -0.149,Y -597.278,Z 272.267,A 0.000,B 0.000,C 90.000,E1 264.090} C_DIS
LIN {X -0.237,Y -599.788,Z 272.254,A 0.000,B 0.000,C 90.000,E1 261.724} C_DIS
LIN {X -0.066,Y -602.982,Z 272.241,A 0.000,B 0.000,C 90.000,E1 259.342} C_DIS
LIN {X 0.066,Y -605.433,Z 272.232,A 0.000,B 0.000,C 90.000,E1 257.757} C_DIS
LIN {X 0.255,Y -607.960,Z 272.223,A 0.000,B 0.000,C 90.000,E1 256.172} C_DIS
LIN {X 0.302,Y -609.988,Z 272.216,A 0.000,B 0.000,C 90.000,E1 254.866} C_DIS
LIN {X -0.121,Y -611.490,Z 272.210,A 0.000,B 0.000,C 90.000,E1 253.866} C_DIS
LIN {X -0.115,Y -612.342,Z 272.206,A 0.000,B 0.000,C 90.000,E1 253.087} C_DIS
LIN {X -0.099,Y -612.919,Z 272.202,A 0.000,B 0.000,C 90.000,E1 252.308} C_DIS
LIN {X 0.143,Y -613.725,Z 272.193,A 0.000,B 0.000,C 90.000,E1 250.732} C_DIS
LIN {X 0.165,Y -613.870,Z 272.189,A 0.000,B 0.000,C 90.000,E1 249.953} C_DIS
LIN {X -0.179,Y -613.843,Z 272.184,A 0.000,B 0.000,C 90.000,E1 249.209} C_DIS
LIN {X 0.055,Y -613.529,Z 272.180,A 0.000,B 0.000,C 90.000,E1 248.411} C_DIS
LIN {X 0.246,Y -612.701,Z 272.174,A 0.000,B 0.000,C 90.000,E1 247.358} C_DIS
LIN {X -0.101,Y -611.858,Z 272.170,A 0.000,B 0.000,C 90.000,E1 246.613} C_DIS
LIN {X -0.172,Y -611.155,Z 272.167,A 0.000,B 0.000,C 90.000,E1 246.102} C_DIS
LIN {X 0.019,Y -609.855,Z 272.163,A 0.000,B 0.000,C 90.000,E1 245.305} C_DIS
LIN {X -0.106,Y -608.326,Z 272.159,A 0.000,B 0.000,C 90.000,E1 244.537} C_DIS
LIN {X -0.240,Y -606.602,Z 272.154,A 0.000,B 0.000,C 90.000,E1 243.768} C_DIS
LIN {X 0.033,Y -603.434,Z 272.147,A 0.000,B 0.000,C 90.000,E1 242.436} C_DIS
LIN {X -0.011,Y -600.037,Z 272.140,A 0.000,B 0.000,C 90.000,E1 241.129} C_DIS
LIN {X 0.188,Y -596.491,Z 272.132,A 0.000,B 0.000,C 90.000,E1 239.793} C_DIS
LIN {X 0.122,Y -593.462,Z 272.126,A 0.000,B 0.000,C 90.000,E1 238.742} C_DIS
LIN {X -0.297,Y -589.485,Z 272.119,A 0.000,B 0.000,C 90.000,E1 237.454} C_DIS
LIN {X 0.219,Y -584.327,Z 272.110,A 0.000,B 0.000,C 90.000,E1 235.801} C_DIS
LIN {X 0.307,Y -578.318,Z 272.100,A 0.000,B 0.000,C 90.000,E1 233.909} C_DIS
LIN {X -0.016,Y -573.343,Z 272.091,A 0.000,B 0.000,C 90.000,E1 232.316} C_DIS
LIN {X -0.313,Y -567.414,Z 272.080,A 0.000,B 0.000,C 90.000,E1 230.436} C_DIS
LIN {X 0.077,Y -564.065,Z 272.074,A 0.000,B 0.000,C 90.000,E1 229.299} C_DIS
LIN {X 0.089,Y -559.764,Z 272.066,A 0.000,B 0.000,C 90.000,E1 227.919} C_DIS
LIN {X 0.019,Y -555.417,Z 272.059,A 0.000,B 0.000,C 90.000,E1 226.539} C_DIS
LIN {X 0.276,Y -550.162,Z 272.049,A 0.000,B 0.000,C 90.000,E1 224.838} C_DIS
LIN {X 0.015,Y -545.750,Z 272.042,A 0.000,B 0.000,C 90.000,E1 223.461} C_DIS
LIN {X 0.081,Y -540.465,Z 272.032,A 0.000,B 0.000,C 90.000,E1 221.757} C_DIS
LIN {X 0.084,Y -536.085,Z 272.024,A 0.000,B 0.000,C 90.000,E1 220.334} C_DIS
LIN {X 0.004,Y -530.837,Z 272.015,A 0.000,B 0.000,C 90.000,E1 218.624} C_DIS
LIN {X 0.186,Y -524.772,Z 272.003,A 0.000,B 0.000,C 90.000,E1 216.583} C_DIS
LIN {X -0.061,Y -519.719,Z 271.994,A 0.000,B 0.000,C 90.000,E1 214.865} C_DIS
LIN {X 0.135,Y -514.769,Z 271.984,A 0.000,B 0.000,C 90.000,E1 213.086} C_DIS
LIN {X 0.045,Y -510.780,Z 271.976,A 0.000,B 0.000,C 90.000,E1 211.623} C_DIS
LIN {X 0.105,Y -505.350,Z 271.964,A 0.000,B 0.000,C 90.000,E1 209.539} C_DIS
LIN {X -0.098,Y -500.992,Z 271.954,A 0.000,B 0.000,C 90.000,E1 207.769} C_DIS
LIN {X -0.218,Y -494.233,Z 271.938,A 0.000,B 0.000,C 90.000,E1 204.771} C_DIS
LIN {X -0.151,Y -489.259,Z 271.924,A 0.000,B 0.000,C 90.000,E1 202.333} C_DIS
LIN {X -0.141,Y -484.673,Z 271.910,A 0.000,B 0.000,C 90.000,E1 199.885} C_DIS
LIN {X 0.029,Y -480.473,Z 271.897,A 0.000,B 0.000,C 90.000,E1 197.402} C_DIS
LIN {X 0.129,Y -478.092,Z 271.888,A 0.000,B 0.000,C 90.000,E1 195.843} C_DIS
LIN {X -0.186,Y -473.754,Z 271.871,A 0.000,B 0.000,C 90.000,E1 192.771} C_DIS
LIN {X 0.002,Y -471.823,Z 271.862,A 0.000,B 0.000,C 90.000,E1 191.186} C_DIS
LIN {X -0.023,Y -468.866,Z 271.848,A 0.000,B 0.000,C 90.000,E1 188.681} C_DIS
LIN {X -0.093,Y -466.619,Z 271.836,A 0.000,B 0.000,C 90.000,E1 186.486} C_DIS
LIN {X -0.065,Y -464.858,Z 271.826,A 0.000,B 0.000,C 90.000,E1 184.588} C_DIS
LIN {X -0.145,Y -462.895,Z 271.811,A 0.000,B 0.000,C 90.000,E1 182.064} C_DIS
LIN {X -0.088,Y -461.064,Z 271.796,A 0.000,B 0.000,C 90.000,E1 179.198} C_DIS
LIN {X 0.186,Y -459.887,Z 271.781,A 0.000,B 0.000,C 90.000,E1 176.617} C_DIS
LIN {X -0.010,Y -459.156,Z 271.767,A 0.000,B 0.000,C 90.000,E1 174.090} C_DIS
LIN {X 0.137,Y -458.914,Z 271.755,A 0.000,B 0.000,C 90.000,E1 171.837} C_DIS
LIN {X 0.121,Y -458.877,Z 271.741,A 0.000,B 0.000,C 90.000,E1 169.285} C_DIS
LIN {X 0.038,Y -459.253,Z 271.728,A 0.000,B 0.000,C 90.000,E1 167.061} C_DIS
LIN {X 0.058,Y -459.636,Z 271.719,A 0.000,B 0.000,C 90.000,E1 165.463} C_DIS
LIN {X 0.161,Y -461.240,Z 271.700,A 0.000,B 0.000,C 90.000,E1 161.945} C_DIS
LIN {X 0.189,Y -463.361,Z 271.684,A 0.000,B 0.000,C 90.000,E1 159.082} C_DIS
LIN {X 0.147,Y -465.311,Z 271.672,A 0.000,B 0.000,C 90.000,E1 156.869} C_DIS
LIN {X 0.032,Y -468.001,Z 271.658,A 0.000,B 0.000,C 90.000,E1 154.357} C_DIS
LIN {X -0.012,Y -471.274,Z 271.644,A 0.000,B 0.000,C 90.000,E1 151.847} C_DIS
LIN {X -0.089,Y -474.499,Z 271.631,A 0.000,B 0.000,C 90.000,E1 149.665} C_DIS
LIN {X 0.168,Y -477.955,Z 271.619,A 0.000,B 0.000,C 90.000,E1 147.454} C_DIS
LIN {X -0.027,Y -481.629,Z 271.607,A 0.000,B 0.000,C 90.000,E1 145.308} C_DIS
LIN {X -0.060,Y -484.810,Z 271.597,A 0.000,B 0.000,C 90.000,E1 143.463} C_DIS
LIN {X 0.141,Y -487.304,Z 271.589,A 0.000,B 0.000,C 90.000,E1 141.904} C_DIS
LIN {X -0.224,Y -489.215,Z 271.582,A 0.000,B 0.000,C 90.000,E1 140.723} C_DIS
LIN {X 0.128,Y -490.931,Z 271.575,A 0.000,B 0.000,C 90.000,E1 139.461} C_DIS
LIN {X -0.034,Y -492.144,Z 271.570,A 0.000,B 0.000,C 90.000,E1 138.566} C_DIS
LIN {X 0.314,Y -493.440,Z 271.563,A 0.000,B 0.000,C 90.000,E1 137.310} C_DIS
LIN {X -0.031,Y -493.983,Z 271.560,A 0.000,B 0.000,C 90.000,E1 136.743} C_DIS
LIN {X 0.170,Y -494.613,Z 271.555,A 0.000,B 0.000,C 90.000,E1 135.810} C_DIS
LIN {X 0.205,Y -494.998,Z 271.548,A 0.000,B 0.000,C 90.000,E1 134.595} C_DIS
LIN {X 0.058,Y -495.073,Z 271.543,A 0.000,B 0.000,C 90.000,E1 133.704} C_DIS
LIN {X 0.270,Y -494.914,Z 271.538,A 0.000,B 0.000,C 90.000,E1 132.771} C_DIS
LIN {X -0.218,Y -494.558,Z 271.533,A 0.000,B 0.000,C 90.000,E1 131.919} C_DIS
LIN {X -0.014,Y -493.901,Z 271.528,A 0.000,B 0.000,C 90.000,E1 130.987} C_DIS
LIN {X -0.141,Y -493.027,Z 271.523,A 0.000,B 0.000,C 90.000,E1 130.092} C_DIS
LIN {X 0.112,Y -491.310,Z 271.514,A 0.000,B 0.000,C 90.000,E1 128.543} C_DIS
LIN {X -0.203,Y -489.654,Z 271.507,A 0.000,B 0.000,C 90.000,E1 127.363} C_DIS
LIN {X 0.235,Y -487.855,Z 271.501,A 0.000,B 0.000,C 90.000,E1 126.091} C_DIS
LIN {X -0.205,Y -485.255,Z 271.492,A 0.000,B 0.000,C 90.000,E1 124.612} C_DIS
LIN {X 0.109,Y -482.469,Z 271.484,A 0.000,B 0.000,C 90.000,E1 123.038} C_DIS
LIN {X -0.086,Y -479.059,Z 271.473,A 0.000,B 0.000,C 90.000,E1 121.209} C_DIS
LIN {X -0.148,Y -476.221,Z 271.465,A 0.000,B 0.000,C 90.000,E1 119.667} C_DIS
LIN {X 0.087,Y -472.739,Z 271.454,A 0.000,B 0.000,C 90.000,E1 117.769} C_DIS
LIN {X -0.140,Y -469.842,Z 271.446,A 0.000,B 0.000,C 90.000,E1 116.232} C_DIS
LIN {X 0.001,Y -466.907,Z 271.437,A 0.000,B 0.000,C 90.000,E1 114.643} C_DIS
LIN {X -0.174,Y -463.406,Z 271.426,A 0.000,B 0.000,C 90.000,E1 112.770} C_DIS
LIN {X 0.147,Y -461.180,Z 271.419,A 0.000,B 0.000,C 90.000,E1 111.461} C_DIS
LIN {X -0.089,Y -459.473,Z 271.414,A 0.000,B 0.000,C 90.000,E1 110.536} C_DIS
LIN {X 0.075,Y -457.804,Z 271.408,A 0.000,B 0.000,C 90.000,E1 109.504} C_DIS
LIN {X 0.035,Y -457.810,Z 271.408,A 0.000,B 0.000,C 90.000,E1 109.504} C_DIS
LIN {X 0.038,Y -466.450,Z 271.386,A 0.000,B 0.000,C 90.000,E1 105.426} C_DIS
LIN {X 0.214,Y -467.944,Z 271.382,A 0.000,B 0.000,C 90.000,E1 104.773} C_DIS
LIN {X 0.179,Y -476.161,Z 271.356,A 0.000,B 0.000,C 90.000,E1 100.074} C_DIS
LIN {X -0.090,Y -482.071,Z 271.330,A 0.000,B 0.000,C 90.000,E1 95.454} C_DIS
LIN {X 0.185,Y -485.495,Z 271.305,A 0.000,B 0.000,C 90.000,E1 90.802} C_DIS
LIN {X 0.218,Y -486.385,Z 271.281,A 0.000,B 0.000,C 90.000,E1 86.502} C_DIS
LIN {X 0.042,Y -486.362,Z 271.279,A 0.000,B 0.000,C 90.000,E1 86.216} C_DIS
LIN {X 0.126,Y -484.687,Z 271.253,A 0.000,B 0.000,C 90.000,E1 81.602} C_DIS
LIN {X 0.025,Y -480.614,Z 271.228,A 0.000,B 0.000,C 90.000,E1 76.992} C_DIS
LIN {X -0.117,Y -480.266,Z 271.226,A 0.000,B 0.000,C 90.000,E1 76.700} C_DIS
LIN {X 0.239,Y -474.093,Z 271.200,A 0.000,B 0.000,C 90.000,E1 72.000} C_DIS
LIN {X 0.076,Y -470.089,Z 271.189,A 0.000,B 0.000,C 90.000,E1 69.934} C_DIS
LIN {X 0.036,Y -470.097,Z 271.189,A 0.000,B 0.000,C 90.000,E1 69.934} C_DIS
LIN {X -0.088,Y -474.295,Z 271.179,A 0.000,B 0.000,C 90.000,E1 68.284} C_DIS
LIN {X -0.047,Y -479.149,Z 271.169,A 0.000,B 0.000,C 90.000,E1 66.410} C_DIS
LIN {X -0.082,Y -481.640,Z 271.164,A 0.000,B 0.000,C 90.000,E1 65.485} C_DIS
LIN {X -0.109,Y -487.462,Z 271.152,A 0.000,B 0.000,C 90.000,E1 63.332} C_DIS
LIN {X 0.050,Y -494.347,Z 271.138,A 0.000,B 0.000,C 90.000,E1 60.873} C_DIS
LIN {X 0.187,Y -500.481,Z 271.127,A 0.000,B 0.000,C 90.000,E1 58.742} C_DIS
LIN {X 0.135,Y -504.877,Z 271.118,A 0.000,B 0.000,C 90.000,E1 57.248} C_DIS
LIN {X -0.260,Y -509.080,Z 271.110,A 0.000,B 0.000,C 90.000,E1 55.801} C_DIS
LIN {X -0.121,Y -511.508,Z 271.105,A 0.000,B 0.000,C 90.000,E1 54.895} C_DIS
LIN {X -0.107,Y -515.344,Z 271.097,A 0.000,B 0.000,C 90.000,E1 53.417} C_DIS
LIN {X 0.284,Y -518.834,Z 271.089,A 0.000,B 0.000,C 90.000,E1 51.904} C_DIS
LIN {X -0.072,Y -521.948,Z 271.080,A 0.000,B 0.000,C 90.000,E1 50.481} C_DIS
LIN {X 0.073,Y -524.159,Z 271.074,A 0.000,B 0.000,C 90.000,E1 49.299} C_DIS
LIN {X -0.109,Y -525.645,Z 271.069,A 0.000,B 0.000,C 90.000,E1 48.447} C_DIS
LIN {X 0.115,Y -526.886,Z 271.064,A 0.000,B 0.000,C 90.000,E1 47.553} C_DIS
LIN {X -0.042,Y -528.005,Z 271.059,A 0.000,B 0.000,C 90.000,E1 46.701} C_DIS
LIN {X 0.179,Y -528.900,Z 271.055,A 0.000,B 0.000,C 90.000,E1 45.810} C_DIS
LIN {X -0.008,Y -529.890,Z 271.048,A 0.000,B 0.000,C 90.000,E1 44.676} C_DIS
LIN {X 0.235,Y -530.374,Z 271.043,A 0.000,B 0.000,C 90.000,E1 43.785} C_DIS
LIN {X -0.301,Y -530.721,Z 271.037,A 0.000,B 0.000,C 90.000,E1 42.690} C_DIS
LIN {X 0.336,Y -530.903,Z 271.032,A 0.000,B 0.000,C 90.000,E1 41.757} C_DIS
LIN {X 0.221,Y -530.924,Z 271.027,A 0.000,B 0.000,C 90.000,E1 40.906} C_DIS
LIN {X -0.240,Y -530.777,Z 271.023,A 0.000,B 0.000,C 90.000,E1 40.092} C_DIS
LIN {X 0.048,Y -530.465,Z 271.018,A 0.000,B 0.000,C 90.000,E1 39.197} C_DIS
LIN {X 0.293,Y -529.664,Z 271.010,A 0.000,B 0.000,C 90.000,E1 37.729} C_DIS
LIN {X 0.220,Y -528.803,Z 271.003,A 0.000,B 0.000,C 90.000,E1 36.583} C_DIS
LIN {X 0.130,Y -527.751,Z 270.997,A 0.000,B 0.000,C 90.000,E1 35.438} C_DIS
LIN {X 0.123,Y -526.197,Z 270.989,A 0.000,B 0.000,C 90.000,E1 33.992} C_DIS
LIN {X 0.091,Y -524.497,Z 270.981,A 0.000,B 0.000,C 90.000,E1 32.546} C_DIS
LIN {X -0.256,Y -522.753,Z 270.973,A 0.000,B 0.000,C 90.000,E1 31.131} C_DIS
LIN {X -0.129,Y -520.253,Z 270.962,A 0.000,B 0.000,C 90.000,E1 29.077} C_DIS
LIN {X 0.005,Y -518.189,Z 270.952,A 0.000,B 0.000,C 90.000,E1 27.308} C_DIS
LIN {X 0.092,Y -515.510,Z 270.939,A 0.000,B 0.000,C 90.000,E1 24.951} C_DIS
LIN {X -0.094,Y -513.742,Z 270.929,A 0.000,B 0.000,C 90.000,E1 23.206} C_DIS
LIN {X 0.277,Y -511.708,Z 270.917,A 0.000,B 0.000,C 90.000,E1 21.099} C_DIS
LIN {X -0.251,Y -509.913,Z 270.906,A 0.000,B 0.000,C 90.000,E1 19.087} C_DIS
LIN {X 0.075,Y -508.060,Z 270.893,A 0.000,B 0.000,C 90.000,E1 16.677} C_DIS
LIN {X 0.108,Y -506.569,Z 270.881,A 0.000,B 0.000,C 90.000,E1 14.592} C_DIS
LIN {X -0.039,Y -505.716,Z 270.873,A 0.000,B 0.000,C 90.000,E1 13.119} C_DIS
LIN {X 0.235,Y -504.925,Z 270.863,A 0.000,B 0.000,C 90.000,E1 11.299} C_DIS
LIN {X 0.179,Y -504.129,Z 270.850,A 0.000,B 0.000,C 90.000,E1 8.916} C_DIS
LIN {X -0.034,Y -503.807,Z 270.836,A 0.000,B 0.000,C 90.000,E1 6.549} C_DIS
LIN {X 0.005,Y -503.930,Z 270.820,A 0.000,B 0.000,C 90.000,E1 3.555} C_DIS
LIN {X -0.157,Y -504.947,Z 270.802,A 0.000,B 0.000,C 90.000,E1 0.286} C_DIS
LIN {X -0.228,Y -506.910,Z 270.784,A 0.000,B 0.000,C 90.000,E1 357.135} C_DIS
LIN {X 0.064,Y -509.041,Z 270.771,A 0.000,B 0.000,C 90.000,E1 354.723} C_DIS
LIN {X 0.206,Y -510.561,Z 270.763,A 0.000,B 0.000,C 90.000,E1 353.223} C_DIS
LIN {X 0.149,Y -514.773,Z 270.746,A 0.000,B 0.000,C 90.000,E1 350.274} C_DIS
LIN {X 0.025,Y -519.568,Z 270.733,A 0.000,B 0.000,C 90.000,E1 347.937} C_DIS
LIN {X -0.205,Y -526.219,Z 270.718,A 0.000,B 0.000,C 90.000,E1 345.338} C_DIS
LIN {X 0.004,Y -529.244,Z 270.712,A 0.000,B 0.000,C 90.000,E1 344.157} C_DIS
LIN {X 0.065,Y -537.145,Z 270.696,A 0.000,B 0.000,C 90.000,E1 341.275} C_DIS
LIN {X -0.224,Y -544.254,Z 270.683,A 0.000,B 0.000,C 90.000,E1 339.028} C_DIS
LIN {X -0.189,Y -550.866,Z 270.672,A 0.000,B 0.000,C 90.000,E1 337.050} C_DIS
LIN {X -0.053,Y -556.728,Z 270.663,A 0.000,B 0.000,C 90.000,E1 335.357} C_DIS
LIN {X -0.132,Y -565.803,Z 270.649,A 0.000,B 0.000,C 90.000,E1 332.871} C_DIS
LIN {X -0.276,Y -570.937,Z 270.642,A 0.000,B 0.000,C 90.000,E1 331.513} C_DIS
LIN {X -0.054,Y -575.806,Z 270.634,A 0.000,B 0.000,C 90.000,E1 330.127} C_DIS
LIN {X 0.256,Y -580.514,Z 270.627,A 0.000,B 0.000,C 90.000,E1 328.742} C_DIS
LIN {X -0.126,Y -588.019,Z 270.615,A 0.000,B 0.000,C 90.000,E1 326.628} C_DIS
LIN {X -0.067,Y -594.012,Z 270.606,A 0.000,B 0.000,C 90.000,E1 325.022} C_DIS
LIN {X -0.120,Y -599.000,Z 270.598,A 0.000,B 0.000,C 90.000,E1 323.703} C_DIS
LIN {X -0.240,Y -601.857,Z 270.594,A 0.000,B 0.000,C 90.000,E1 322.924} C_DIS
LIN {X -0.294,Y -606.314,Z 270.587,A 0.000,B 0.000,C 90.000,E1 321.618} C_DIS
LIN {X -0.079,Y -611.481,Z 270.578,A 0.000,B 0.000,C 90.000,E1 320.033} C_DIS
LIN {X 0.018,Y -615.613,Z 270.571,A 0.000,B 0.000,C 90.000,E1 318.728} C_DIS
LIN {X -0.344,Y -619.738,Z 270.564,A 0.000,B 0.000,C 90.000,E1 317.472} C_DIS
LIN {X -0.062,Y -622.983,Z 270.558,A 0.000,B 0.000,C 90.000,E1 316.419} C_DIS
LIN {X 0.018,Y -627.357,Z 270.549,A 0.000,B 0.000,C 90.000,E1 314.879} C_DIS
LIN {X -0.032,Y -630.213,Z 270.544,A 0.000,B 0.000,C 90.000,E1 313.866} C_DIS
LIN {X -0.036,Y -632.932,Z 270.538,A 0.000,B 0.000,C 90.000,E1 312.852} C_DIS
LIN {X -0.004,Y -635.420,Z 270.532,A 0.000,B 0.000,C 90.000,E1 311.838} C_DIS
LIN {X 0.160,Y -637.127,Z 270.528,A 0.000,B 0.000,C 90.000,E1 311.067} C_DIS
LIN {X -0.077,Y -638.693,Z 270.524,A 0.000,B 0.000,C 90.000,E1 310.334} C_DIS
LIN {X 0.115,Y -640.119,Z 270.520,A 0.000,B 0.000,C 90.000,E1 309.564} C_DIS
LIN {X 0.314,Y -641.745,Z 270.514,A 0.000,B 0.000,C 90.000,E1 308.543} C_DIS
LIN {X 0.029,Y -643.243,Z 270.509,A 0.000,B 0.000,C 90.000,E1 307.569} C_DIS
LIN {X -0.123,Y -644.543,Z 270.503,A 0.000,B 0.000,C 90.000,E1 306.583} C_DIS
LIN {X 0.229,Y -645.201,Z 270.499,A 0.000,B 0.000,C 90.000,E1 305.804} C_DIS
LIN {X 0.108,Y -645.667,Z 270.494,A 0.000,B 0.000,C 90.000,E1 304.818} C_DIS
LIN {X -0.013,Y -645.816,Z 270.488,A 0.000,B 0.000,C 90.000,E1 303.833} C_DIS
LIN {X -0.014,Y -645.822,Z 270.484,A 0.000,B 0.000,C 90.000,E1 303.086} C_DIS
LIN {X -0.014,Y -645.531,Z 270.480,A 0.000,B 0.000,C 90.000,E1 302.339} C_DIS
LIN {X -0.017,Y -644.915,Z 270.476,A 0.000,B 0.000,C 90.000,E1 301.592} C_DIS
LIN {X -0.029,Y -643.940,Z 270.471,A 0.000,B 0.000,C 90.000,E1 300.846} C_DIS
LIN {X 0.177,Y -642.667,Z 270.467,A 0.000,B 0.000,C 90.000,E1 300.079} C_DIS
LIN {X 0.201,Y -640.587,Z 270.462,A 0.000,B 0.000,C 90.000,E1 299.077} C_DIS
LIN {X -0.115,Y -638.246,Z 270.456,A 0.000,B 0.000,C 90.000,E1 298.103} C_DIS
LIN {X 0.157,Y -635.087,Z 270.449,A 0.000,B 0.000,C 90.000,E1 296.821} C_DIS
LIN {X -0.193,Y -631.770,Z 270.442,A 0.000,B 0.000,C 90.000,E1 295.591} C_DIS
LIN {X -0.262,Y -627.029,Z 270.432,A 0.000,B 0.000,C 90.000,E1 293.823} C_DIS
LIN {X 0.117,Y -623.674,Z 270.425,A 0.000,B 0.000,C 90.000,E1 292.514} C_DIS
LIN {X -0.070,Y -618.499,Z 270.414,A 0.000,B 0.000,C 90.000,E1 290.482} C_DIS
LIN {X 0.019,Y -614.169,Z 270.404,A 0.000,B 0.000,C 90.000,E1 288.671} C_DIS
LIN {X 0.008,Y -608.498,Z 270.389,A 0.000,B 0.000,C 90.000,E1 286.079} C_DIS
LIN {X 0.161,Y -604.022,Z 270.376,A 0.000,B 0.000,C 90.000,E1 283.716} C_DIS
LIN {X -0.209,Y -599.290,Z 270.359,A 0.000,B 0.000,C 90.000,E1 280.602} C_DIS
LIN {X -0.213,Y -596.029,Z 270.343,A 0.000,B 0.000,C 90.000,E1 277.701} C_DIS
LIN {X -0.262,Y -594.545,Z 270.332,A 0.000,B 0.000,C 90.000,E1 275.853} C_DIS
LIN {X -0.118,Y -593.148,Z 270.316,A 0.000,B 0.000,C 90.000,E1 272.922} C_DIS
LIN {X 0.119,Y -592.834,Z 270.299,A 0.000,B 0.000,C 90.000,E1 269.714} C_DIS
LIN {X 0.174,Y -593.820,Z 270.282,A 0.000,B 0.000,C 90.000,E1 266.788} C_DIS
LIN {X 0.087,Y -595.833,Z 270.268,A 0.000,B 0.000,C 90.000,E1 264.147} C_DIS
LIN {X -0.041,Y -598.330,Z 270.254,A 0.000,B 0.000,C 90.000,E1 261.781} C_DIS
LIN {X 0.089,Y -601.538,Z 270.241,A 0.000,B 0.000,C 90.000,E1 259.398} C_DIS
LIN {X 0.068,Y -604.005,Z 270.232,A 0.000,B 0.000,C 90.000,E1 257.825} C_DIS
LIN {X 0.095,Y -606.954,Z 270.222,A 0.000,B 0.000,C 90.000,E1 255.992} C_DIS
LIN {X -0.032,Y -608.946,Z 270.215,A 0.000,B 0.000,C 90.000,E1 254.700} C_DIS
LIN {X -0.309,Y -610.428,Z 270.209,A 0.000,B 0.000,C 90.000,E1 253.685} C_DIS
LIN {X -0.312,Y -611.209,Z 270.205,A 0.000,B 0.000,C 90.000,E1 252.906} C_DIS
LIN {X 0.209,Y -611.853,Z 270.199,A 0.000,B 0.000,C 90.000,E1 251.819} C_DIS
LIN {X 0.165,Y -612.368,Z 270.193,A 0.000,B 0.000,C 90.000,E1 250.786} C_DIS
LIN {X 0.128,Y -612.560,Z 270.188,A 0.000,B 0.000,C 90.000,E1 249.752} C_DIS
LIN {X 0.351,Y -612.464,Z 270.183,A 0.000,B 0.000,C 90.000,E1 248.954} C_DIS
LIN {X -0.222,Y -612.071,Z 270.179,A 0.000,B 0.000,C 90.000,E1 248.230} C_DIS
LIN {X -0.053,Y -611.154,Z 270.173,A 0.000,B 0.000,C 90.000,E1 247.177} C_DIS
LIN {X -0.173,Y -610.256,Z 270.169,A 0.000,B 0.000,C 90.000,E1 246.410} C_DIS
LIN {X 0.014,Y -609.055,Z 270.165,A 0.000,B 0.000,C 90.000,E1 245.613} C_DIS
LIN {X -0.117,Y -607.632,Z 270.160,A 0.000,B 0.000,C 90.000,E1 244.845} C_DIS
LIN {X 0.236,Y -605.339,Z 270.154,A 0.000,B 0.000,C 90.000,E1 243.768} C_DIS
LIN {X -0.049,Y -602.202,Z 270.147,A 0.000,B 0.000,C 90.000,E1 242.487} C_DIS
LIN {X -0.034,Y -599.478,Z 270.141,A 0.000,B 0.000,C 90.000,E1 241.435} C_DIS
LIN {X -0.135,Y -595.951,Z 270.134,A 0.000,B 0.000,C 90.000,E1 240.127} C_DIS
LIN {X -0.205,Y -592.964,Z 270.128,A 0.000,B 0.000,C 90.000,E1 239.076} C_DIS
LIN {X -0.014,Y -589.785,Z 270.122,A 0.000,B 0.000,C 90.000,E1 237.995} C_DIS
LIN {X 0.131,Y -586.444,Z 270.116,A 0.000,B 0.000,C 90.000,E1 236.914} C_DIS
LIN {X 0.095,Y -581.248,Z 270.107,A 0.000,B 0.000,C 90.000,E1 235.308} C_DIS
LIN {X 0.109,Y -575.321,Z 270.097,A 0.000,B 0.000,C 90.000,E1 233.417} C_DIS
LIN {X -0.102,Y -572.009,Z 270.091,A 0.000,B 0.000,C 90.000,E1 232.351} C_DIS
LIN {X -0.084,Y -566.104,Z 270.080,A 0.000,B 0.000,C 90.000,E1 230.436} C_DIS
LIN {X 0.287,Y -562.743,Z 270.074,A 0.000,B 0.000,C 90.000,E1 229.299} C_DIS
LIN {X -0.101,Y -558.432,Z 270.066,A 0.000,B 0.000,C 90.000,E1 227.957} C_DIS
LIN {X 0.178,Y -554.086,Z 270.059,A 0.000,B 0.000,C 90.000,E1 226.539} C_DIS
LIN {X 0.016,Y -548.806,Z 270.049,A 0.000,B 0.000,C 90.000,E1 224.879} C_DIS
LIN {X 0.120,Y -544.383,Z 270.042,A 0.000,B 0.000,C 90.000,E1 223.461} C_DIS
LIN {X 0.165,Y -538.231,Z 270.031,A 0.000,B 0.000,C 90.000,E1 221.472} C_DIS
LIN {X 0.062,Y -532.905,Z 270.021,A 0.000,B 0.000,C 90.000,E1 219.769} C_DIS
LIN {X 0.006,Y -528.530,Z 270.013,A 0.000,B 0.000,C 90.000,E1 218.338} C_DIS
LIN {X 0.131,Y -522.520,Z 270.002,A 0.000,B 0.000,C 90.000,E1 216.297} C_DIS
LIN {X -0.095,Y -516.657,Z 269.990,A 0.000,B 0.000,C 90.000,E1 214.278} C_DIS
LIN {X -0.039,Y -510.974,Z 269.979,A 0.000,B 0.000,C 90.000,E1 212.212} C_DIS
LIN {X 0.023,Y -505.443,Z 269.967,A 0.000,B 0.000,C 90.000,E1 210.129} C_DIS
LIN {X 0.118,Y -500.305,Z 269.956,A 0.000,B 0.000,C 90.000,E1 208.025} C_DIS
LIN {X -0.032,Y -493.461,Z 269.939,A 0.000,B 0.000,C 90.000,E1 205.027} C_DIS
LIN {X 0.016,Y -488.474,Z 269.926,A 0.000,B 0.000,C 90.000,E1 202.589} C_DIS
LIN {X 0.164,Y -484.421,Z 269.914,A 0.000,B 0.000,C 90.000,E1 200.429} C_DIS
LIN {X -0.135,Y -480.136,Z 269.900,A 0.000,B 0.000,C 90.000,E1 198.000} C_DIS
LIN {X -0.068,Y -477.273,Z 269.890,A 0.000,B 0.000,C 90.000,E1 196.134} C_DIS
LIN {X 0.040,Y -472.887,Z 269.872,A 0.000,B 0.000,C 90.000,E1 193.008} C_DIS
LIN {X 0.213,Y -470.958,Z 269.864,A 0.000,B 0.000,C 90.000,E1 191.422} C_DIS
LIN {X 0.166,Y -467.967,Z 269.850,A 0.000,B 0.000,C 90.000,E1 188.916} C_DIS
LIN {X -0.123,Y -465.366,Z 269.836,A 0.000,B 0.000,C 90.000,E1 186.429} C_DIS
LIN {X -0.121,Y -463.636,Z 269.825,A 0.000,B 0.000,C 90.000,E1 184.531} C_DIS
LIN {X -0.237,Y -461.689,Z 269.811,A 0.000,B 0.000,C 90.000,E1 182.007} C_DIS
LIN {X -0.220,Y -459.902,Z 269.795,A 0.000,B 0.000,C 90.000,E1 179.141} C_DIS
LIN {X 0.207,Y -458.613,Z 269.779,A 0.000,B 0.000,C 90.000,E1 176.216} C_DIS
LIN {X 0.009,Y -457.980,Z 269.765,A 0.000,B 0.000,C 90.000,E1 173.685} C_DIS
LIN {X -0.101,Y -457.824,Z 269.754,A 0.000,B 0.000,C 90.000,E1 171.781} C_DIS
LIN {X 0.151,Y -457.803,Z 269.742,A 0.000,B 0.000,C 90.000,E1 169.511} C_DIS
LIN {X -0.047,Y -458.169,Z 269.729,A 0.000,B 0.000,C 90.000,E1 167.297} C_DIS
LIN {X -0.049,Y -458.563,Z 269.721,A 0.000,B 0.000,C 90.000,E1 165.700} C_DIS
LIN {X -0.077,Y -460.277,Z 269.699,A 0.000,B 0.000,C 90.000,E1 161.873} C_DIS
LIN {X -0.234,Y -462.451,Z 269.683,A 0.000,B 0.000,C 90.000,E1 159.028} C_DIS
LIN {X -0.194,Y -464.733,Z 269.669,A 0.000,B 0.000,C 90.000,E1 156.485} C_DIS
LIN {X -0.035,Y -468.332,Z 269.652,A 0.000,B 0.000,C 90.000,E1 153.307} C_DIS
LIN {X 0.005,Y -471.333,Z 269.639,A 0.000,B 0.000,C 90.000,E1 151.101} C_DIS
LIN {X 0.169,Y -474.138,Z 269.629,A 0.000,B 0.000,C 90.000,E1 149.203} C_DIS
LIN {X -0.179,Y -477.137,Z 269.619,A 0.000,B 0.000,C 90.000,E1 147.375} C_DIS
LIN {X 0.003,Y -480.851,Z 269.607,A 0.000,B 0.000,C 90.000,E1 145.182} C_DIS
LIN {X 0.128,Y -483.481,Z 269.598,A 0.000,B 0.000,C 90.000,E1 143.623} C_DIS
LIN {X 0.124,Y -486.463,Z 269.588,A 0.000,B 0.000,C 90.000,E1 141.778} C_DIS
LIN {X 0.053,Y -488.362,Z 269.581,A 0.000,B 0.000,C 90.000,E1 140.561} C_DIS
LIN {X 0.229,Y -490.442,Z 269.573,A 0.000,B 0.000,C 90.000,E1 139.013} C_DIS
LIN {X 0.224,Y -491.211,Z 269.569,A 0.000,B 0.000,C 90.000,E1 138.405} C_DIS
LIN {X 0.028,Y -492.181,Z 269.564,A 0.000,B 0.000,C 90.000,E1 137.514} C_DIS
LIN {X -0.127,Y -493.002,Z 269.559,A 0.000,B 0.000,C 90.000,E1 136.620} C_DIS
LIN {X 0.222,Y -493.478,Z 269.556,A 0.000,B 0.000,C 90.000,E1 135.972} C_DIS
LIN {X 0.239,Y -493.876,Z 269.549,A 0.000,B 0.000,C 90.000,E1 134.757} C_DIS
LIN {X 0.081,Y -494.017,Z 269.544,A 0.000,B 0.000,C 90.000,E1 133.866} C_DIS
LIN {X -0.239,Y -493.818,Z 269.537,A 0.000,B 0.000,C 90.000,E1 132.690} C_DIS
LIN {X -0.041,Y -493.444,Z 269.532,A 0.000,B 0.000,C 90.000,E1 131.757} C_DIS
LIN {X 0.148,Y -492.763,Z 269.527,A 0.000,B 0.000,C 90.000,E1 130.825} C_DIS
LIN {X 0.007,Y -491.882,Z 269.522,A 0.000,B 0.000,C 90.000,E1 129.930} C_DIS
LIN {X 0.083,Y -490.522,Z 269.515,A 0.000,B 0.000,C 90.000,E1 128.705} C_DIS
LIN {X -0.238,Y -488.947,Z 269.508,A 0.000,B 0.000,C 90.000,E1 127.523} C_DIS
LIN {X -0.202,Y -487.165,Z 269.502,A 0.000,B 0.000,C 90.000,E1 126.297} C_DIS
LIN {X -0.027,Y -485.654,Z 269.496,A 0.000,B 0.000,C 90.000,E1 125.358} C_DIS
LIN {X 0.067,Y -483.517,Z 269.490,A 0.000,B 0.000,C 90.000,E1 124.119} C_DIS
LIN {X -0.110,Y -480.165,Z 269.479,A 0.000,B 0.000,C 90.000,E1 122.291} C_DIS
LIN {X 0.098,Y -477.361,Z 269.471,A 0.000,B 0.000,C 90.000,E1 120.718} C_DIS
LIN {X -0.014,Y -475.051,Z 269.464,A 0.000,B 0.000,C 90.000,E1 119.489} C_DIS
LIN {X -0.216,Y -471.591,Z 269.453,A 0.000,B 0.000,C 90.000,E1 117.641} C_DIS
LIN {X -0.041,Y -468.701,Z 269.445,A 0.000,B 0.000,C 90.000,E1 116.052} C_DIS
LIN {X 0.022,Y -465.173,Z 269.434,A 0.000,B 0.000,C 90.000,E1 114.155} C_DIS
LIN {X -0.047,Y -462.890,Z 269.427,A 0.000,B 0.000,C 90.000,E1 112.898} C_DIS
LIN {X 0.189,Y -460.057,Z 269.418,A 0.000,B 0.000,C 90.000,E1 111.280} C_DIS
LIN {X -0.112,Y -457.400,Z 269.410,A 0.000,B 0.000,C 90.000,E1 109.758} C_DIS
LIN {X -0.152,Y -457.400,Z 269.410,A 0.000,B 0.000,C 90.000,E1 109.758} C_DIS
LIN {X 0.144,Y -466.111,Z 269.387,A 0.000,B 0.000,C 90.000,E1 105.552} C_DIS
LIN {X -0.132,Y -467.682,Z 269.383,A 0.000,B 0.000,C 90.000,E1 104.954} C_DIS
LIN {X -0.175,Y -475.895,Z 269.357,A 0.000,B 0.000,C 90.000,E1 100.254} C_DIS
LIN {X 0.133,Y -476.346,Z 269.355,A 0.000,B 0.000,C 90.000,E1 99.905} C_DIS
LIN {X 0.089,Y -481.860,Z 269.331,A 0.000,B 0.000,C 90.000,E1 95.568} C_DIS
LIN {X -0.064,Y -482.189,Z 269.329,A 0.000,B 0.000,C 90.000,E1 95.277} C_DIS
LIN {X -0.130,Y -485.355,Z 269.305,A 0.000,B 0.000,C 90.000,E1 90.974} C_DIS
LIN {X 0.180,Y -485.532,Z 269.304,A 0.000,B 0.000,C 90.000,E1 90.630} C_DIS
LIN {X -0.097,Y -486.341,Z 269.281,A 0.000,B 0.000,C 90.000,E1 86.674} C_DIS
LIN {X 0.036,Y -486.275,Z 269.278,A 0.000,B 0.000,C 90.000,E1 86.045} C_DIS
LIN {X -0.243,Y -484.693,Z 269.254,A 0.000,B 0.000,C 90.000,E1 81.781} C_DIS
LIN {X 0.104,Y -484.547,Z 269.253,A 0.000,B 0.000,C 90.000,E1 81.432} C_DIS
LIN {X -0.026,Y -480.485,Z 269.227,A 0.000,B 0.000,C 90.000,E1 76.825} C_DIS
LIN {X -0.129,Y -474.242,Z 269.201,A 0.000,B 0.000,C 90.000,E1 72.181} C_DIS
LIN {X -0.162,Y -473.756,Z 269.199,A 0.000,B 0.000,C 90.000,E1 71.873} C_DIS
LIN {X -0.084,Y -469.739,Z 269.188,A 0.000,B 0.000,C 90.000,E1 69.752} C_DIS
LIN {X -0.123,Y -469.747,Z 269.187,A 0.000,B 0.000,C 90.000,E1 69.752} C_DIS
LIN {X -0.057,Y -473.890,Z 269.178,A 0.000,B 0.000,C 90.000,E1 68.103} C_DIS
LIN {X -0.043,Y -479.605,Z 269.166,A 0.000,B 0.000,C 90.000,E1 65.921} C_DIS
LIN {X -0.117,Y -486.244,Z 269.153,A 0.000,B 0.000,C 90.000,E1 63.461} C_DIS
LIN {X -0.011,Y -492.192,Z 269.141,A 0.000,B 0.000,C 90.000,E1 61.307} C_DIS
LIN {X -0.045,Y -496.542,Z 269.132,A 0.000,B 0.000,C 90.000,E1 59.793} C_DIS
LIN {X -0.137,Y -501.855,Z 269.122,A 0.000,B 0.000,C 90.000,E1 57.995} C_DIS
LIN {X -0.084,Y -504.444,Z 269.117,A 0.000,B 0.000,C 90.000,E1 57.089} C_DIS
LIN {X -0.061,Y -508.660,Z 269.109,A 0.000,B 0.000,C 90.000,E1 55.595} C_DIS
LIN {X -0.099,Y -512.558,Z 269.101,A 0.000,B 0.000,C 90.000,E1 54.116} C_DIS
LIN {X 0.077,Y -514.852,Z 269.096,A 0.000,B 0.000,C 90.000,E1 53.210} C_DIS
LIN {X 0.049,Y -518.276,Z 269.088,A 0.000,B 0.000,C 90.000,E1 51.743} C_DIS
LIN {X 0.088,Y -521.328,Z 269.079,A 0.000,B 0.000,C 90.000,E1 50.275} C_DIS
LIN {X -0.226,Y -523.987,Z 269.071,A 0.000,B 0.000,C 90.000,E1 48.852} C_DIS
LIN {X -0.022,Y -525.375,Z 269.066,A 0.000,B 0.000,C 90.000,E1 47.957} C_DIS
LIN {X 0.116,Y -526.821,Z 269.060,A 0.000,B 0.000,C 90.000,E1 46.782} C_DIS
LIN {X 0.321,Y -527.725,Z 269.055,A 0.000,B 0.000,C 90.000,E1 45.891} C_DIS
LIN {X 0.118,Y -528.702,Z 269.049,A 0.000,B 0.000,C 90.000,E1 44.757} C_DIS
LIN {X -0.074,Y -529.369,Z 269.042,A 0.000,B 0.000,C 90.000,E1 43.623} C_DIS
LIN {X 0.094,Y -529.729,Z 269.034,A 0.000,B 0.000,C 90.000,E1 42.162} C_DIS
LIN {X -0.053,Y -529.765,Z 269.028,A 0.000,B 0.000,C 90.000,E1 41.024} C_DIS
LIN {X -0.177,Y -529.625,Z 269.023,A 0.000,B 0.000,C 90.000,E1 40.172} C_DIS
LIN {X 0.098,Y -529.296,Z 269.018,A 0.000,B 0.000,C 90.000,E1 39.277} C_DIS
LIN {X -0.093,Y -528.521,Z 269.010,A 0.000,B 0.000,C 90.000,E1 37.855} C_DIS
LIN {X 0.235,Y -527.642,Z 269.004,A 0.000,B 0.000,C 90.000,E1 36.664} C_DIS
LIN {X 0.133,Y -526.573,Z 268.997,A 0.000,B 0.000,C 90.000,E1 35.518} C_DIS
LIN {X -0.293,Y -525.297,Z 268.991,A 0.000,B 0.000,C 90.000,E1 34.405} C_DIS
LIN {X 0.101,Y -523.581,Z 268.983,A 0.000,B 0.000,C 90.000,E1 32.911} C_DIS
LIN {X 0.019,Y -521.819,Z 268.975,A 0.000,B 0.000,C 90.000,E1 31.465} C_DIS
LIN {X -0.258,Y -519.596,Z 268.965,A 0.000,B 0.000,C 90.000,E1 29.745} C_DIS
LIN {X -0.129,Y -517.533,Z 268.955,A 0.000,B 0.000,C 90.000,E1 27.975} C_DIS
LIN {X -0.290,Y -515.442,Z 268.946,A 0.000,B 0.000,C 90.000,E1 26.232} C_DIS
LIN {X 0.070,Y -513.231,Z 268.934,A 0.000,B 0.000,C 90.000,E1 24.131} C_DIS
LIN {X 0.189,Y -511.754,Z 268.926,A 0.000,B 0.000,C 90.000,E1 22.642} C_DIS
LIN {X -0.158,Y -509.747,Z 268.914,A 0.000,B 0.000,C 90.000,E1 20.610} C_DIS
LIN {X 0.193,Y -508.492,Z 268.906,A 0.000,B 0.000,C 90.000,E1 19.087} C_DIS
LIN {X -0.097,Y -506.829,Z 268.895,A 0.000,B 0.000,C 90.000,E1 17.040} C_DIS
LIN {X -0.090,Y -505.283,Z 268.883,A 0.000,B 0.000,C 90.000,E1 14.954} C_DIS
LIN {X -0.197,Y -504.193,Z 268.873,A 0.000,B 0.000,C 90.000,E1 13.175} C_DIS
LIN {X -0.061,Y -503.393,Z 268.863,A 0.000,B 0.000,C 90.000,E1 11.366} C_DIS
LIN {X -0.134,Y -502.475,Z 268.848,A 0.000,B 0.000,C 90.000,E1 8.681} C_DIS
LIN {X 0.170,Y -502.224,Z 268.837,A 0.000,B 0.000,C 90.000,E1 6.549} C_DIS
LIN {X -0.230,Y -502.242,Z 268.822,A 0.000,B 0.000,C 90.000,E1 3.898} C_DIS
LIN {X -0.241,Y -502.890,Z 268.807,A 0.000,B 0.000,C 90.000,E1 1.203} C_DIS
LIN {X -0.143,Y -503.970,Z 268.794,A 0.000,B 0.000,C 90.000,E1 358.912} C_DIS
LIN {X 0.138,Y -505.448,Z 268.782,A 0.000,B 0.000,C 90.000,E1 356.788} C_DIS
LIN {X -0.044,Y -507.325,Z 268.771,A 0.000,B 0.000,C 90.000,E1 354.723} C_DIS
LIN {X 0.067,Y -508.813,Z 268.762,A 0.000,B 0.000,C 90.000,E1 353.223} C_DIS
LIN {X -0.085,Y -513.617,Z 268.744,A 0.000,B 0.000,C 90.000,E1 349.982} C_DIS
LIN {X -0.242,Y -518.644,Z 268.731,A 0.000,B 0.000,C 90.000,E1 347.645} C_DIS
LIN {X -0.008,Y -524.620,Z 268.718,A 0.000,B 0.000,C 90.000,E1 345.283} C_DIS
LIN {X 0.173,Y -527.687,Z 268.712,A 0.000,B 0.000,C 90.000,E1 344.102} C_DIS
LIN {X 0.172,Y -535.604,Z 268.696,A 0.000,B 0.000,C 90.000,E1 341.221} C_DIS
LIN {X -0.147,Y -540.010,Z 268.688,A 0.000,B 0.000,C 90.000,E1 339.826} C_DIS
LIN {X 0.032,Y -547.486,Z 268.675,A 0.000,B 0.000,C 90.000,E1 337.539} C_DIS
LIN {X -0.124,Y -553.297,Z 268.666,A 0.000,B 0.000,C 90.000,E1 335.869} C_DIS
LIN {X 0.005,Y -558.256,Z 268.658,A 0.000,B 0.000,C 90.000,E1 334.460} C_DIS
LIN {X -0.148,Y -565.419,Z 268.647,A 0.000,B 0.000,C 90.000,E1 332.538} C_DIS
LIN {X -0.117,Y -569.553,Z 268.641,A 0.000,B 0.000,C 90.000,E1 331.435} C_DIS
LIN {X -0.199,Y -574.441,Z 268.634,A 0.000,B 0.000,C 90.000,E1 330.078} C_DIS
LIN {X 0.378,Y -579.169,Z 268.626,A 0.000,B 0.000,C 90.000,E1 328.663} C_DIS
LIN {X -0.214,Y -585.759,Z 268.616,A 0.000,B 0.000,C 90.000,E1 326.834} C_DIS
LIN {X 0.283,Y -591.809,Z 268.607,A 0.000,B 0.000,C 90.000,E1 325.182} C_DIS
LIN {X -0.065,Y -597.789,Z 268.598,A 0.000,B 0.000,C 90.000,E1 323.623} C_DIS
LIN {X -0.195,Y -600.616,Z 268.594,A 0.000,B 0.000,C 90.000,E1 322.844} C_DIS
LIN {X -0.268,Y -605.023,Z 268.586,A 0.000,B 0.000,C 90.000,E1 321.537} C_DIS
LIN {X 0.117,Y -609.329,Z 268.579,A 0.000,B 0.000,C 90.000,E1 320.194} C_DIS
LIN {X -0.284,Y -613.537,Z 268.572,A 0.000,B 0.000,C 90.000,E1 318.933} C_DIS
LIN {X -0.382,Y -618.579,Z 268.563,A 0.000,B 0.000,C 90.000,E1 317.391} C_DIS
LIN {X 0.335,Y -621.846,Z 268.557,A 0.000,B 0.000,C 90.000,E1 316.296} C_DIS
LIN {X -0.059,Y -626.248,Z 268.549,A 0.000,B 0.000,C 90.000,E1 314.798} C_DIS
LIN {X -0.248,Y -629.789,Z 268.542,A 0.000,B 0.000,C 90.000,E1 313.542} C_DIS
LIN {X -0.260,Y -632.434,Z 268.536,A 0.000,B 0.000,C 90.000,E1 312.528} C_DIS
LIN {X 0.129,Y -635.419,Z 268.529,A 0.000,B 0.000,C 90.000,E1 311.229} C_DIS
LIN {X -0.228,Y -637.458,Z 268.524,A 0.000,B 0.000,C 90.000,E1 310.253} C_DIS
LIN {X -0.050,Y -638.860,Z 268.519,A 0.000,B 0.000,C 90.000,E1 309.483} C_DIS
LIN {X -0.267,Y -640.074,Z 268.515,A 0.000,B 0.000,C 90.000,E1 308.749} C_DIS
LIN {X 0.334,Y -641.897,Z 268.508,A 0.000,B 0.000,C 90.000,E1 307.443} C_DIS
LIN {X 0.143,Y -642.876,Z 268.504,A 0.000,B 0.000,C 90.000,E1 306.710} C_DIS
LIN {X -0.012,Y -643.712,Z 268.499,A 0.000,B 0.000,C 90.000,E1 305.724} C_DIS
LIN {X -0.040,Y -644.084,Z 268.494,A 0.000,B 0.000,C 90.000,E1 304.978} C_DIS
LIN {X 0.307,Y -644.235,Z 268.490,A 0.000,B 0.000,C 90.000,E1 304.199} C_DIS
LIN {X -0.188,Y -644.310,Z 268.485,A 0.000,B 0.000,C 90.000,E1 303.245} C_DIS
LIN {X 0.148,Y -644.072,Z 268.480,A 0.000,B 0.000,C 90.000,E1 302.467} C_DIS
LIN {X 0.129,Y -643.488,Z 268.476,A 0.000,B 0.000,C 90.000,E1 301.720} C_DIS
LIN {X -0.294,Y -642.969,Z 268.474,A 0.000,B 0.000,C 90.000,E1 301.258} C_DIS
LIN {X 0.227,Y -641.802,Z 268.469,A 0.000,B 0.000,C 90.000,E1 300.463} C_DIS
LIN {X 0.238,Y -639.882,Z 268.464,A 0.000,B 0.000,C 90.000,E1 299.461} C_DIS
LIN {X -0.037,Y -637.043,Z 268.457,A 0.000,B 0.000,C 90.000,E1 298.231} C_DIS
LIN {X -0.352,Y -633.875,Z 268.450,A 0.000,B 0.000,C 90.000,E1 297.001} C_DIS
LIN {X -0.156,Y -630.549,Z 268.443,A 0.000,B 0.000,C 90.000,E1 295.720} C_DIS
LIN {X -0.252,Y -625.789,Z 268.433,A 0.000,B 0.000,C 90.000,E1 293.951} C_DIS
LIN {X 0.108,Y -622.459,Z 268.426,A 0.000,B 0.000,C 90.000,E1 292.642} C_DIS
LIN {X -0.108,Y -617.256,Z 268.414,A 0.000,B 0.000,C 90.000,E1 290.610} C_DIS
LIN {X 0.154,Y -612.934,Z 268.404,A 0.000,B 0.000,C 90.000,E1 288.779} C_DIS
LIN {X -0.087,Y -607.250,Z 268.390,A 0.000,B 0.000,C 90.000,E1 286.205} C_DIS
LIN {X 0.140,Y -603.702,Z 268.380,A 0.000,B 0.000,C 90.000,E1 284.356} C_DIS
LIN {X 0.040,Y -598.344,Z 268.361,A 0.000,B 0.000,C 90.000,E1 280.950} C_DIS
LIN {X -0.285,Y -595.210,Z 268.346,A 0.000,B 0.000,C 90.000,E1 278.341} C_DIS
LIN {X 0.270,Y -592.725,Z 268.329,A 0.000,B 0.000,C 90.000,E1 275.106} C_DIS
LIN {X 0.106,Y -591.575,Z 268.314,A 0.000,B 0.000,C 90.000,E1 272.465} C_DIS
LIN {X 0.117,Y -591.655,Z 268.293,A 0.000,B 0.000,C 90.000,E1 268.740} C_DIS
LIN {X -0.227,Y -593.261,Z 268.275,A 0.000,B 0.000,C 90.000,E1 265.584} C_DIS
LIN {X -0.221,Y -595.723,Z 268.261,A 0.000,B 0.000,C 90.000,E1 262.932} C_DIS
LIN {X 0.246,Y -600.095,Z 268.242,A 0.000,B 0.000,C 90.000,E1 259.454} C_DIS
LIN {X 0.199,Y -602.560,Z 268.233,A 0.000,B 0.000,C 90.000,E1 257.881} C_DIS
LIN {X 0.050,Y -605.529,Z 268.223,A 0.000,B 0.000,C 90.000,E1 256.061} C_DIS
LIN {X 0.049,Y -607.534,Z 268.215,A 0.000,B 0.000,C 90.000,E1 254.755} C_DIS
LIN {X -0.244,Y -609.046,Z 268.210,A 0.000,B 0.000,C 90.000,E1 253.740} C_DIS
LIN {X -0.259,Y -609.840,Z 268.205,A 0.000,B 0.000,C 90.000,E1 252.960} C_DIS
LIN {X 0.247,Y -610.492,Z 268.199,A 0.000,B 0.000,C 90.000,E1 251.873} C_DIS
LIN {X -0.073,Y -611.076,Z 268.192,A 0.000,B 0.000,C 90.000,E1 250.604} C_DIS
LIN {X -0.076,Y -611.216,Z 268.188,A 0.000,B 0.000,C 90.000,E1 249.826} C_DIS
LIN {X 0.129,Y -611.131,Z 268.184,A 0.000,B 0.000,C 90.000,E1 249.028} C_DIS
LIN {X -0.236,Y -610.758,Z 268.179,A 0.000,B 0.000,C 90.000,E1 248.284} C_DIS
LIN {X -0.081,Y -609.838,Z 268.174,A 0.000,B 0.000,C 90.000,E1 247.230} C_DIS
LIN {X 0.105,Y -608.946,Z 268.169,A 0.000,B 0.000,C 90.000,E1 246.433} C_DIS
LIN {X 0.013,Y -608.179,Z 268.166,A 0.000,B 0.000,C 90.000,E1 245.921} C_DIS
LIN {X -0.127,Y -606.828,Z 268.162,A 0.000,B 0.000,C 90.000,E1 245.153} C_DIS
LIN {X 0.325,Y -605.809,Z 268.159,A 0.000,B 0.000,C 90.000,E1 244.588} C_DIS
LIN {X -0.100,Y -604.066,Z 268.155,A 0.000,B 0.000,C 90.000,E1 243.845} C_DIS
LIN {X -0.069,Y -601.590,Z 268.149,A 0.000,B 0.000,C 90.000,E1 242.794} C_DIS
LIN {X 0.187,Y -598.922,Z 268.143,A 0.000,B 0.000,C 90.000,E1 241.719} C_DIS
LIN {X 0.272,Y -594.705,Z 268.134,A 0.000,B 0.000,C 90.000,E1 240.127} C_DIS
LIN {X 0.076,Y -590.883,Z 268.127,A 0.000,B 0.000,C 90.000,E1 238.820} C_DIS
LIN {X -0.265,Y -587.669,Z 268.121,A 0.000,B 0.000,C 90.000,E1 237.788} C_DIS
LIN {X 0.033,Y -583.352,Z 268.114,A 0.000,B 0.000,C 90.000,E1 236.421} C_DIS
LIN {X -0.232,Y -577.341,Z 268.103,A 0.000,B 0.000,C 90.000,E1 234.562} C_DIS
LIN {X 0.020,Y -571.506,Z 268.092,A 0.000,B 0.000,C 90.000,E1 232.637} C_DIS
LIN {X -0.092,Y -566.443,Z 268.083,A 0.000,B 0.000,C 90.000,E1 231.009} C_DIS
LIN {X 0.026,Y -562.270,Z 268.076,A 0.000,B 0.000,C 90.000,E1 229.622} C_DIS
LIN {X 0.000,Y -557.981,Z 268.068,A 0.000,B 0.000,C 90.000,E1 228.243} C_DIS
LIN {X -0.070,Y -552.735,Z 268.059,A 0.000,B 0.000,C 90.000,E1 226.581} C_DIS
LIN {X -0.247,Y -547.434,Z 268.049,A 0.000,B 0.000,C 90.000,E1 224.919} C_DIS
LIN {X -0.162,Y -542.096,Z 268.040,A 0.000,B 0.000,C 90.000,E1 223.218} C_DIS
LIN {X -0.173,Y -535.938,Z 268.029,A 0.000,B 0.000,C 90.000,E1 221.229} C_DIS
LIN {X 0.050,Y -528.878,Z 268.016,A 0.000,B 0.000,C 90.000,E1 218.910} C_DIS
LIN {X 0.219,Y -523.645,Z 268.007,A 0.000,B 0.000,C 90.000,E1 217.156} C_DIS
LIN {X 0.004,Y -519.405,Z 267.999,A 0.000,B 0.000,C 90.000,E1 215.724} C_DIS
END
